# B&R Automation Studio project EFI (part 3)

### Hardware
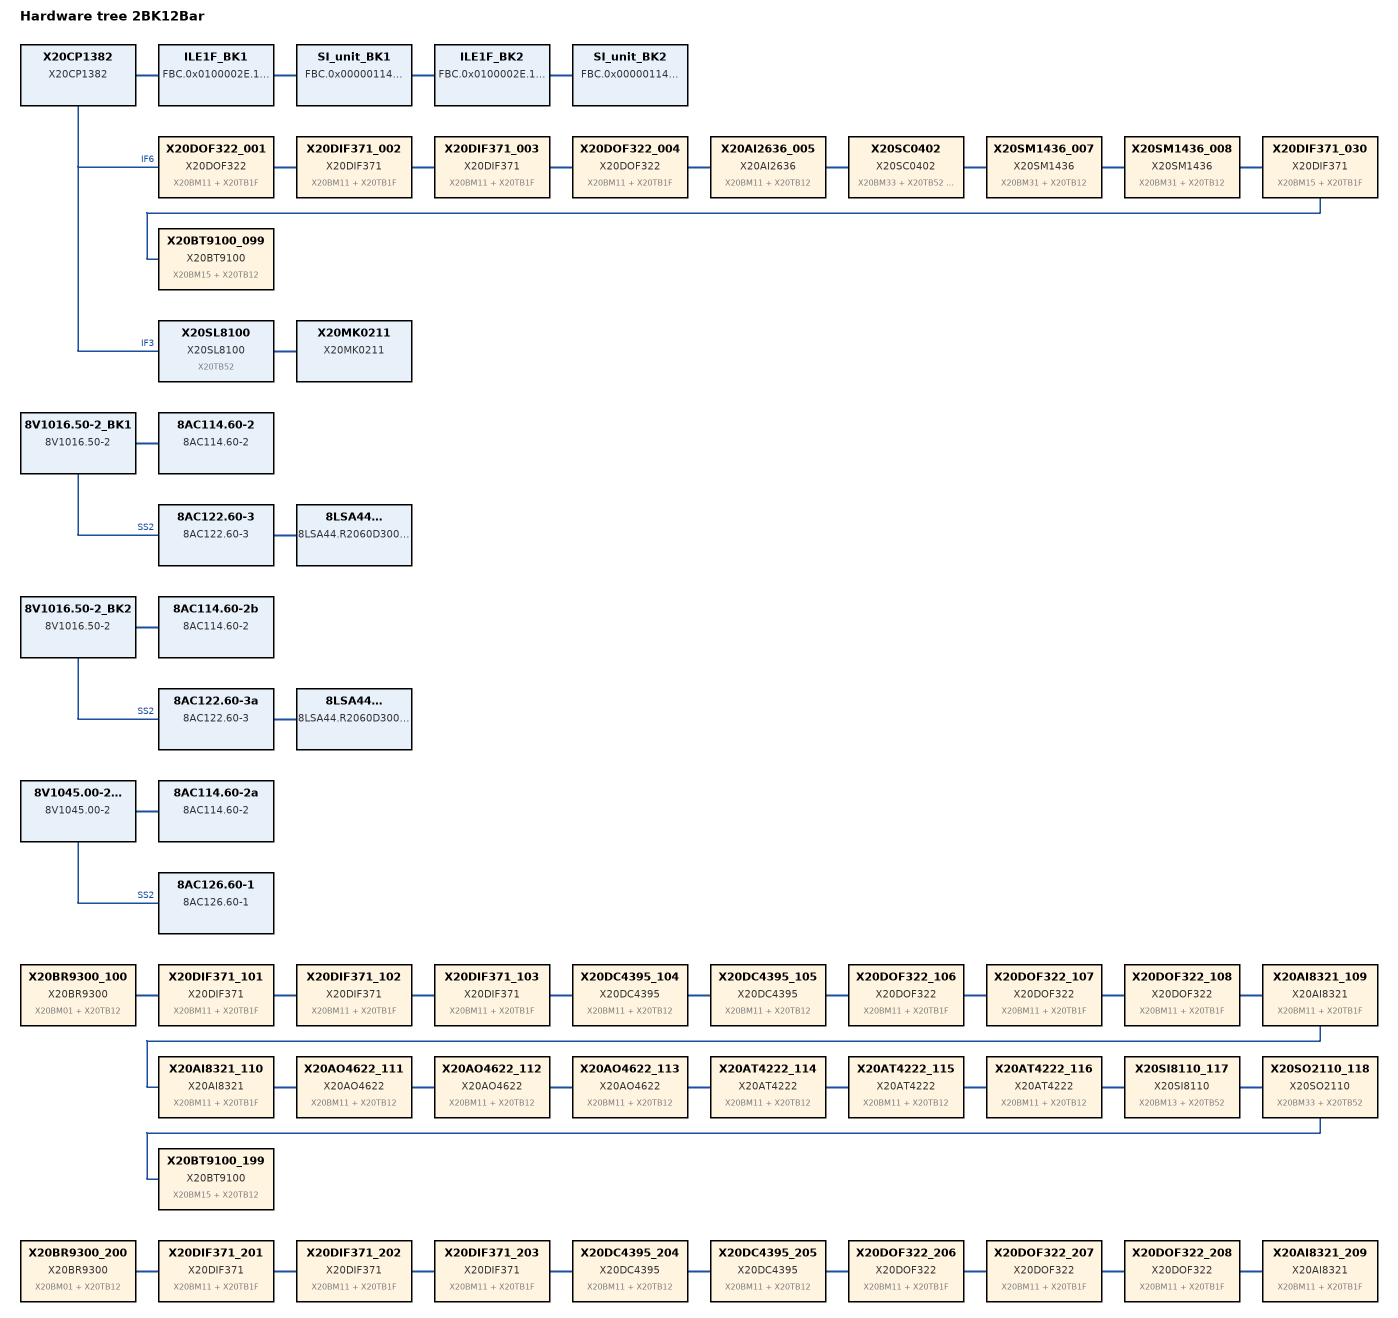
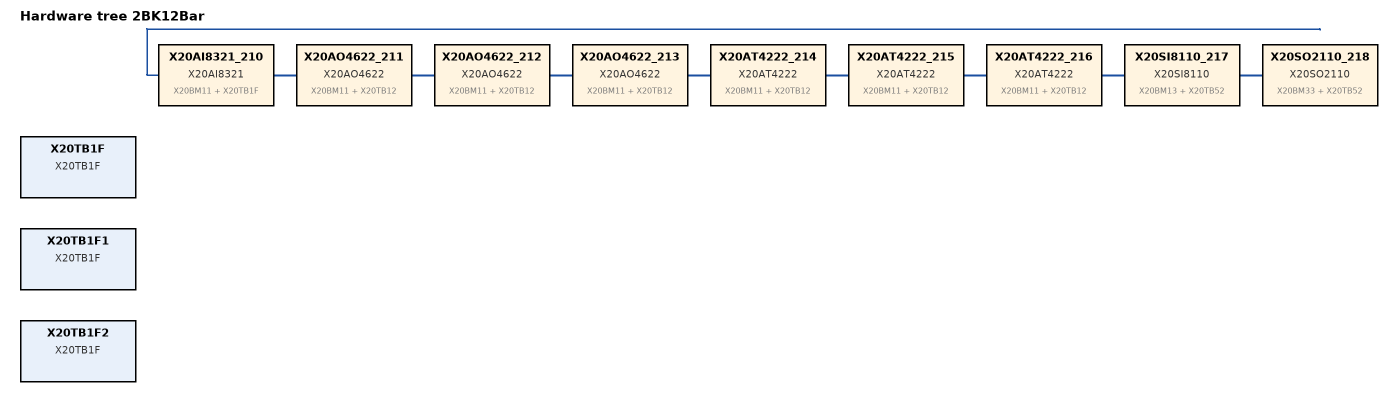
```
8AC114.60-2 : 8AC114.60-2 v1.0.0.8  [SS -> 8V1016.50-2_BK1.SS1; PLK1 -> 8AC114.60-2a.PLK2 (NodeNumber=2) [Cable Type=PowerlinkCable, Length=10, Version=1.0.0.3]; PLK2 -> 8AC114.60-2b.PLK1 (NodeNumber=2) [Cable Type=PowerlinkCable, Length=10, Version=1.0.0.3]]
8AC114.60-2a : 8AC114.60-2 v1.0.0.8  [SS -> 8V1045.00-2_BELT.SS1; PLK1 -> X20SL8100.PLK2 (NodeNumber=1) [Cable Type=PowerlinkCable, Length=10, Version=1.0.0.3]; PLK2 -> 8AC114.60-2.PLK1 (NodeNumber=1) [Cable Type=PowerlinkCable, Length=10, Version=1.0.0.3]]
8AC114.60-2b : 8AC114.60-2 v1.0.0.8  [SS -> 8V1016.50-2_BK2.SS1; PLK1 -> 8AC114.60-2.PLK2 (NodeNumber=3) [Cable Type=PowerlinkCable, Length=10, Version=1.0.0.3]]
8AC122.60-3 : 8AC122.60-3 v2.2.0.0  [SS -> 8V1016.50-2_BK1.SS2]
8AC122.60-3a : 8AC122.60-3 v2.2.0.0  [SS -> 8V1016.50-2_BK2.SS2]
8AC126.60-1 : 8AC126.60-1 v2.2.0.0  [SS -> 8V1045.00-2_BELT.SS2]
8LSA44.R2060D300-3 : 8LSA44.R2060D300-3 v2.2.0.0  [EC -> 8AC122.60-3.EC; MT -> 8V1016.50-2_BK1.MT1]
8LSA44.R2060D300-3a : 8LSA44.R2060D300-3 v2.2.0.0  [EC -> 8AC122.60-3a.EC; MT -> 8V1016.50-2_BK2.MT1]
8V1016.50-2_BK1 : 8V1016.50-2 v2.2.0.0
  SinglePhaseOperation = on
  BothEndSwitchesAreNormallyOpen_r1 = on
  QuickStopIsNormallyOpen_r1 = on
8V1016.50-2_BK2 : 8V1016.50-2 v2.2.0.0
  SinglePhaseOperation = on
  BothEndSwitchesAreNormallyOpen_r1 = on
  QuickStopIsNormallyOpen_r1 = on
8V1045.00-2_BELT : 8V1045.00-2 v2.2.0.0
ILE1F_BK1 : FBC.0x0100002E.1.SEILE1F_0110E v1.10 (OrderNumber=ILE1F)  [CAN1 -> X20CP1382.IF7 (NodeNumber=5)]
  p1403_transmissionselection = 1
  plifeguarding_guardtime = 500
  plifeguarding_retryfactor = 10
  p3001_parametername = mandatory
  p3001_objecttype = 9
  p3001_subnumber = 0x3
  p3001_parametervalue = 
  p3001_objflags = 0
  p3001sub0_parametername = number of entries
  p3001sub0_objecttype = 7
  p3001sub0_datatype = 5
  p3001sub0_accesstype = ro
  p3001sub0_pdomapping = 0
  p3001sub1_parametername = Config.PrgNo
  p3001sub1_objecttype = 7
  p3001sub1_datatype = 7
  p3001sub1_lowlimit = 
  p3001sub1_highlimit = 
  p3001sub1_accesstype = ro
  p3001sub1_pdomapping = 0
  p3001sub2_parametername = Config.PrgVer
  p3001sub2_objecttype = 7
  p3001sub2_datatype = 7
  p3001sub2_lowlimit = 
  p3001sub2_highlimit = 
  p3001sub2_accesstype = ro
  p3001sub2_pdomapping = 0
  p300b_parametername = system settings
  p300b_objecttype = 9
  p300b_subnumber = 0x7
  p300b_parametervalue = 
  p300b_objflags = 0
  p300bsub0_parametername = number of entries
  p300bsub0_objecttype = 7
  p300bsub0_datatype = 5
  p300bsub0_accesstype = ro
  p300bsub0_pdomapping = 0
  p300bsub1_parametername = Settings.name1
  p300bsub1_objecttype = 7
  p300bsub1_datatype = 7
  p300bsub1_lowlimit = 
  p300bsub1_highlimit = 
  p300bsub1_accesstype = rw
  p300bsub1_pdomapping = 0
  p300bsub1_parametervalue = 
  p300bsub1_objflags = 0
  p300bsub2_parametername = Settings.name2
  p300bsub2_objecttype = 7
  p300bsub2_datatype = 7
  p300bsub2_lowlimit = 
  p300bsub2_highlimit = 
  p300bsub2_accesstype = rw
  p300bsub2_pdomapping = 0
  p300bsub2_parametervalue = 
  p300bsub2_objflags = 0
  p300bsub6_parametername = Commands.eeprSave
  p300bsub6_objecttype = 7
  p300bsub6_datatype = 6
  p300bsub6_lowlimit = 
  p300bsub6_highlimit = 
  p300bsub6_accesstype = rw
  p300bsub6_pdomapping = 0
  p300bsub6_parametervalue = 1
  p300bsub6_objflags = 0
  p300bsub7_parametername = Commands.stateSave
  p300bsub7_objecttype = 7
  p300bsub7_datatype = 6
  p300bsub7_lowlimit = 
  p300bsub7_highlimit = 
  p300bsub7_accesstype = ro
  p300bsub7_pdomapping = 0
  p300bsub8_parametername = Commands.default
  p300bsub8_objecttype = 7
  p300bsub8_datatype = 6
  p300bsub8_lowlimit = 
  p300bsub8_highlimit = 
  p300bsub8_accesstype = rw
  p300bsub8_pdomapping = 0
  p300bsub8_parametervalue = 
  p300bsub8_objflags = 0
  p300bsub9_parametername = Commands.stateDef
  p300bsub9_objecttype = 7
  p300bsub9_datatype = 6
  p300bsub9_lowlimit = 
  p300bsub9_highlimit = 
  p300bsub9_accesstype = ro
  p300bsub9_pdomapping = 0
  p300f_parametername = controller  settings
  p300f_objecttype = 9
  p300f_subnumber = 0xE
  p300f_parametervalue = 
  p300f_objflags = 0
  p300fsub0_parametername = number of entries
  p300fsub0_objecttype = 7
  p300fsub0_datatype = 5
  p300fsub0_accesstype = ro
  p300fsub0_pdomapping = 0
  p300fsub1_parametername = Config.I_nomDrv
  p300fsub1_objecttype = 7
  p300fsub1_datatype = 6
  p300fsub1_accesstype = ro
  p300fsub1_pdomapping = 0
  p300fsub2_parametername = Config.I_maxDrv
  p300fsub2_objecttype = 7
  p300fsub2_datatype = 6
  p300fsub2_accesstype = ro
  p300fsub2_pdomapping = 0
  p300fsub3_parametername = Settings.I_max
  p300fsub3_objecttype = 7
  p300fsub3_datatype = 6
  p300fsub3_accesstype = rw
  p300fsub3_pdomapping = 0
  p300fsub3_parametervalue = 60
  p300fsub3_objflags = 0
  p300fsub5_parametername = Settings.I_maxBlk
  p300fsub5_objecttype = 7
  p300fsub5_datatype = 6
  p300fsub5_lowlimit = 
  p300fsub5_highlimit = 
  p300fsub5_accesstype = rw
  p300fsub5_pdomapping = 0
  p300fsub5_parametervalue = 20
  p300fsub5_objflags = 0
  p300fsub7_parametername = Settings.p_maxDiff
  p300fsub7_objecttype = 7
  p300fsub7_datatype = 6
  p300fsub7_lowlimit = 
  p300fsub7_highlimit = 
  p300fsub7_accesstype = rw
  p300fsub7_pdomapping = 0
  p300fsub7_parametervalue = 24
  p300fsub7_objflags = 0
  p300fsub8_parametername = Control.KPn
  p300fsub8_objecttype = 7
  p300fsub8_datatype = 6
  p300fsub8_lowlimit = 
  p300fsub8_highlimit = 
  p300fsub8_accesstype = rw
  p300fsub8_pdomapping = 0
  p300fsub8_parametervalue = 60
  p300fsub8_objflags = 0
  p300fsub9_parametername = Control.TNn
  p300fsub9_objecttype = 7
  p300fsub9_datatype = 6
  p300fsub9_lowlimit = 
  p300fsub9_highlimit = 
  p300fsub9_accesstype = rw
  p300fsub9_pdomapping = 0
  p300fsub9_parametervalue = 10000
  p300fsub9_objflags = 0
  p300fsuba_parametername = Control.KPp
  p300fsuba_objecttype = 7
  p300fsuba_datatype = 6
  p300fsuba_lowlimit = 
  p300fsuba_highlimit = 
  p300fsuba_accesstype = rw
  p300fsuba_pdomapping = 0
  p300fsuba_parametervalue = 300
  p300fsuba_objflags = 0
  p300fsubb_parametername = Control.KFPp
  p300fsubb_objecttype = 7
  p300fsubb_datatype = 6
  p300fsubb_lowlimit = 
  p300fsubb_highlimit = 
  p300fsubb_accesstype = rw
  p300fsubb_pdomapping = 0
  p300fsubb_parametervalue = 32767
  p300fsubb_objflags = 0
  p300fsubc_parametername = Settings.T_block
  p300fsubc_objecttype = 7
  p300fsubc_datatype = 6
  p300fsubc_lowlimit = 
  p300fsubc_highlimit = 
  p300fsubc_accesstype = rw
  p300fsubc_pdomapping = 0
  p300fsubc_parametervalue = 100
  p300fsubc_objflags = 0
  p300fsubd_parametername = Status.p_difPeak
  p300fsubd_objecttype = 7
  p300fsubd_datatype = 7
  p300fsubd_lowlimit = 
  p300fsubd_highlimit = 
  p300fsubd_accesstype = rw
  p300fsubd_pdomapping = 0
  p300fsubd_parametervalue = 
  p300fsubd_objflags = 0
  p300fsubf_parametername = Settings.p_win
  p300fsubf_objecttype = 7
  p300fsubf_datatype = 6
  p300fsubf_lowlimit = 
  p300fsubf_highlimit = 
  p300fsubf_accesstype = rw
  p300fsubf_pdomapping = 0
  p300fsubf_parametervalue = 1
  p300fsubf_objflags = 0
  p300fsub10_parametername = Settings.p_winTime
  p300fsub10_objecttype = 7
  p300fsub10_datatype = 6
  p300fsub10_lowlimit = 
  p300fsub10_highlimit = 
  p300fsub10_accesstype = rw
  p300fsub10_pdomapping = 0
  p300fsub10_parametervalue = 0
  p300fsub10_objflags = 0
  p3016_parametername = rs485
  p3016_objecttype = 9
  p3016_subnumber = 0x4
  p3016_parametervalue = 
  p3016_objflags = 0
  p3016sub0_parametername = number of entries
  p3016sub0_objecttype = 7
  p3016sub0_datatype = 5
  p3016sub0_accesstype = ro
  p3016sub0_pdomapping = 0
  p3016sub1_parametername = RS485.serBaud
  p3016sub1_objecttype = 7
  p3016sub1_datatype = 6
  p3016sub1_lowlimit = 
  p3016sub1_highlimit = 
  p3016sub1_accesstype = rw
  p3016sub1_pdomapping = 0
  p3016sub1_parametervalue = 
  p3016sub1_objflags = 0
  p3016sub2_parametername = RS485.serAdr
  p3016sub2_objecttype = 7
  p3016sub2_datatype = 6
  p3016sub2_lowlimit = 
  p3016sub2_highlimit = 
  p3016sub2_accesstype = rw
  p3016sub2_pdomapping = 0
  p3016sub2_parametervalue = 
  p3016sub2_objflags = 0
  p3016sub3_parametername = RS485.serFormat
  p3016sub3_objecttype = 7
  p3016sub3_datatype = 6
  p3016sub3_lowlimit = 
  p3016sub3_highlimit = 
  p3016sub3_accesstype = rw
  p3016sub3_pdomapping = 0
  p3016sub3_parametervalue = 
  p3016sub3_objflags = 0
  p3017_parametername = can
  p3017_objecttype = 9
  p3017_subnumber = 0x3
  p3017_parametervalue = 
  p3017_objflags = 0
  p3017sub0_parametername = number of entries
  p3017sub0_objecttype = 7
  p3017sub0_datatype = 5
  p3017sub0_accesstype = ro
  p3017sub0_pdomapping = 0
  p3017sub2_parametername = CAN.canAddr
  p3017sub2_objecttype = 7
  p3017sub2_datatype = 6
  p3017sub2_lowlimit = 
  p3017sub2_highlimit = 
  p3017sub2_accesstype = rw
  p3017sub2_pdomapping = 0
  p3017sub2_parametervalue = 
  p3017sub2_objflags = 0
  p3017sub3_parametername = CAN.canBaud
  p3017sub3_objecttype = 7
  p3017sub3_datatype = 6
  p3017sub3_lowlimit = 
  p3017sub3_highlimit = 
  p3017sub3_accesstype = rw
  p3017sub3_pdomapping = 0
  p3017sub3_parametervalue = 
  p3017sub3_objflags = 0
  p301c_parametername = settings1
  p301c_objecttype = 9
  p301c_subnumber = 0xF
  p301c_parametervalue = 
  p301c_objflags = 0
  p301csub0_parametername = number of entries
  p301csub0_objecttype = 7
  p301csub0_datatype = 5
  p301csub0_accesstype = ro
  p301csub0_pdomapping = 0
  p301csub3_parametername = Status.xMode_act
  p301csub3_objecttype = 7
  p301csub3_datatype = 6
  p301csub3_lowlimit = 
  p301csub3_highlimit = 
  p301csub3_accesstype = ro
  p301csub3_pdomapping = 0
  p301csub6_parametername = Motion.invertDir
  p301csub6_objecttype = 7
  p301csub6_datatype = 6
  p301csub6_lowlimit = 
  p301csub6_highlimit = 
  p301csub6_accesstype = rw
  p301csub6_pdomapping = 0
  p301csub6_parametervalue = 0
  p301csub6_objflags = 0
  p301csuba_parametername = Status.WarnSig
  p301csuba_objecttype = 7
  p301csuba_datatype = 6
  p301csuba_lowlimit = 
  p301csuba_highlimit = 
  p301csuba_accesstype = ro
  p301csuba_pdomapping = 0
  p301csubb_parametername = Settings.WarnOvrun
  p301csubb_objecttype = 7
  p301csubb_datatype = 6
  p301csubb_lowlimit = 
  p301csubb_highlimit = 
  p301csubb_accesstype = rw
  p301csubb_pdomapping = 0
  p301csubb_parametervalue = 0
  p301csubb_objflags = 0
  p301csubd_parametername = Settings.SignEnabl
  p301csubd_objecttype = 7
  p301csubd_datatype = 6
  p301csubd_lowlimit = 
  p301csubd_highlimit = 
  p301csubd_accesstype = rw
  p301csubd_pdomapping = 0
  p301csubd_parametervalue = 3
  p301csubd_objflags = 0
  p301csube_parametername = Settings.SignLevel
  p301csube_objecttype = 7
  p301csube_datatype = 6
  p301csube_lowlimit = 
  p301csube_highlimit = 
  p301csube_accesstype = rw
  p301csube_pdomapping = 0
  p301csube_parametervalue = 0
  p301csube_objflags = 0
  p301csubf_parametername = Status.Sign_SR
  p301csubf_objecttype = 7
  p301csubf_datatype = 6
  p301csubf_lowlimit = 
  p301csubf_highlimit = 
  p301csubf_accesstype = ro
  p301csubf_pdomapping = 0
  p301csub11_parametername = Status.FltSig
  p301csub11_objecttype = 7
  p301csub11_datatype = 7
  p301csub11_lowlimit = 
  p301csub11_highlimit = 
  p301csub11_accesstype = ro
  p301csub11_pdomapping = 0
  p301csub12_parametername = Status.FltSig_SR
  p301csub12_objecttype = 7
  p301csub12_datatype = 7
  p301csub12_lowlimit = 
  p301csub12_highlimit = 
  p301csub12_accesstype = ro
  p301csub12_pdomapping = 0
  p301csub13_parametername = Status.action_st
  p301csub13_objecttype = 7
  p301csub13_datatype = 6
  p301csub13_lowlimit = 
  p301csub13_highlimit = 
  p301csub13_accesstype = ro
  p301csub13_pdomapping = 0
  p301csub15_parametername = Motion.dec_Stop
  p301csub15_objecttype = 7
  p301csub15_datatype = 7
  p301csub15_lowlimit = 
  p301csub15_highlimit = 
  p301csub15_accesstype = rw
  p301csub15_pdomapping = 0
  p301csub15_parametervalue = 4960
  p301csub15_objflags = 0
  p301csub18_parametername = Settings.Flt_pDiff
  p301csub18_objecttype = 7
  p301csub18_datatype = 6
  p301csub18_lowlimit = 
  p301csub18_highlimit = 
  p301csub18_accesstype = rw
  p301csub18_pdomapping = 0
  p301csub18_parametervalue = 3
  p301csub18_objflags = 0
  p301d_parametername = settings2
  p301d_objecttype = 9
  p301d_subnumber = 0x4
  p301d_parametervalue = 
  p301d_objflags = 0
  p301dsub0_parametername = number of entries
  p301dsub0_objecttype = 7
  p301dsub0_datatype = 5
  p301dsub0_accesstype = ro
  p301dsub0_pdomapping = 0
  p301dsub2_parametername = Config.ResolutM
  p301dsub2_objecttype = 7
  p301dsub2_datatype = 6
  p301dsub2_accesstype = ro
  p301dsub2_pdomapping = 0
  p301dsub17_parametername = Motion.v_target0
  p301dsub17_objecttype = 7
  p301dsub17_datatype = 6
  p301dsub17_accesstype = rw
  p301dsub17_pdomapping = 0
  p301dsub17_parametervalue = 1000
  p301dsub17_objflags = 0
  p301dsub1a_parametername = Motion.acc
  p301dsub1a_objecttype = 7
  p301dsub1a_datatype = 7
  p301dsub1a_lowlimit = 
  p301dsub1a_highlimit = 
  p301dsub1a_accesstype = rw
  p301dsub1a_pdomapping = 0
  p301dsub1a_parametervalue = 2442
  p301dsub1a_objflags = 0
  p301e_parametername = pdo data
  p301e_objecttype = 9
  p301e_subnumber = 0xC
  p301e_parametervalue = 
  p301e_objflags = 0
  p301esub0_parametername = number of entries
  p301esub0_objecttype = 7
  p301esub0_datatype = 5
  p301esub0_accesstype = ro
  p301esub0_pdomapping = 0
  p301esubb_parametername = Status.ModeError
  p301esubb_objecttype = 7
  p301esubb_datatype = 6
  p301esubb_lowlimit = 
  p301esubb_highlimit = 
  p301esubb_accesstype = ro
  p301esubb_pdomapping = 0
  p301f_parametername = status
  p301f_objecttype = 9
  p301f_subnumber = 0x11
  p301f_parametervalue = 
  p301f_objflags = 0
  p301fsub0_parametername = number of entries
  p301fsub0_objecttype = 7
  p301fsub0_datatype = 5
  p301fsub0_accesstype = ro
  p301fsub0_pdomapping = 0
  p301fsub1_parametername = Status.v_ref
  p301fsub1_objecttype = 7
  p301fsub1_datatype = 4
  p301fsub1_lowlimit = 
  p301fsub1_highlimit = 
  p301fsub1_accesstype = ro
  p301fsub1_pdomapping = 0
  p301fsub2_parametername = Status.v_act
  p301fsub2_objecttype = 7
  p301fsub2_datatype = 4
  p301fsub2_lowlimit = 
  p301fsub2_highlimit = 
  p301fsub2_accesstype = ro
  p301fsub2_pdomapping = 0
  p301fsub5_parametername = Status.p_ref
  p301fsub5_objecttype = 7
  p301fsub5_datatype = 4
  p301fsub5_lowlimit = 
  p301fsub5_highlimit = 
  p301fsub5_accesstype = ro
  p301fsub5_pdomapping = 0
  p301fsub6_parametername = Status.p_act
  p301fsub6_objecttype = 7
  p301fsub6_datatype = 4
  p301fsub6_lowlimit = 
  p301fsub6_highlimit = 
  p301fsub6_accesstype = ro
  p301fsub6_pdomapping = 0
  p301fsub7_parametername = Status.p_dif
  p301fsub7_objecttype = 7
  p301fsub7_datatype = 4
  p301fsub7_lowlimit = 
  p301fsub7_highlimit = 
  p301fsub7_accesstype = ro
  p301fsub7_pdomapping = 0
  p301fsub8_parametername = Status.n_ref
  p301fsub8_objecttype = 7
  p301fsub8_datatype = 3
  p301fsub8_lowlimit = 
  p301fsub8_highlimit = 
  p301fsub8_accesstype = ro
  p301fsub8_pdomapping = 0
  p301fsub9_parametername = Status.n_act
  p301fsub9_objecttype = 7
  p301fsub9_datatype = 3
  p301fsub9_lowlimit = 
  p301fsub9_highlimit = 
  p301fsub9_accesstype = ro
  p301fsub9_pdomapping = 0
  p301fsubc_parametername = Status.I_act
  p301fsubc_objecttype = 7
  p301fsubc_datatype = 3
  p301fsubc_lowlimit = 
  p301fsubc_highlimit = 
  p301fsubc_accesstype = ro
  p301fsubc_pdomapping = 0
  p301fsub14_parametername = Status.UDC_act
  p301fsub14_objecttype = 7
  p301fsub14_datatype = 6
  p301fsub14_lowlimit = 
  p301fsub14_highlimit = 
  p301fsub14_accesstype = ro
  p301fsub14_pdomapping = 0
  p301fsub19_parametername = Status.TPA_act
  p301fsub19_objecttype = 7
  p301fsub19_datatype = 6
  p301fsub19_lowlimit = 
  p301fsub19_highlimit = 
  p301fsub19_accesstype = ro
  p301fsub19_pdomapping = 0
  p301fsub1c_parametername = Status.v_pref
  p301fsub1c_objecttype = 7
  p301fsub1c_datatype = 4
  p301fsub1c_lowlimit = 
  p301fsub1c_highlimit = 
  p301fsub1c_accesstype = ro
  p301fsub1c_pdomapping = 0
  p301fsub1e_parametername = Status.p_target
  p301fsub1e_objecttype = 7
  p301fsub1e_datatype = 4
  p301fsub1e_lowlimit = 
  p301fsub1e_highlimit = 
  p301fsub1e_accesstype = ro
  p301fsub1e_pdomapping = 0
  p301fsub1f_parametername = Status.p_profile
  p301fsub1f_objecttype = 7
  p301fsub1f_datatype = 4
  p301fsub1f_lowlimit = 
  p301fsub1f_highlimit = 
  p301fsub1f_accesstype = ro
  p301fsub1f_pdomapping = 0
  p301fsub23_parametername = Status.n_profile
  p301fsub23_objecttype = 7
  p301fsub23_datatype = 3
  p301fsub23_lowlimit = 
  p301fsub23_highlimit = 
  p301fsub23_accesstype = ro
  p301fsub23_pdomapping = 0
  p301fsub26_parametername = Status.n_target
  p301fsub26_objecttype = 7
  p301fsub26_datatype = 3
  p301fsub26_lowlimit = 
  p301fsub26_highlimit = 
  p301fsub26_accesstype = ro
  p301fsub26_pdomapping = 0
  p301fsub2d_parametername = Status.n_pref
  p301fsub2d_objecttype = 7
  p301fsub2d_datatype = 3
  p301fsub2d_lowlimit = 
  p301fsub2d_highlimit = 
  p301fsub2d_accesstype = ro
  p301fsub2d_pdomapping = 0
  p3020_parametername = error
  p3020_objecttype = 9
  p3020_subnumber = 0x5
  p3020_parametervalue = 
  p3020_objflags = 0
  p3020sub0_parametername = number of entries
  p3020sub0_objecttype = 7
  p3020sub0_datatype = 5
  p3020sub0_accesstype = ro
  p3020sub0_pdomapping = 0
  p3020sub1_parametername = ErrorMemAvailable
  p3020sub1_objecttype = 7
  p3020sub1_datatype = 6
  p3020sub1_lowlimit = 
  p3020sub1_highlimit = 
  p3020sub1_accesstype = ro
  p3020sub1_pdomapping = 0
  p3020sub2_parametername = Commands.del_err
  p3020sub2_objecttype = 7
  p3020sub2_datatype = 6
  p3020sub2_lowlimit = 
  p3020sub2_highlimit = 
  p3020sub2_accesstype = rw
  p3020sub2_pdomapping = 0
  p3020sub2_parametervalue = 
  p3020sub2_objflags = 0
  p3020sub6_parametername = PowerOnCount
  p3020sub6_objecttype = 7
  p3020sub6_datatype = 7
  p3020sub6_lowlimit = 
  p3020sub6_highlimit = 
  p3020sub6_accesstype = ro
  p3020sub6_pdomapping = 0
  p3020sub7_parametername = Status.StopFault
  p3020sub7_objecttype = 7
  p3020sub7_datatype = 6
  p3020sub7_lowlimit = 
  p3020sub7_highlimit = 
  p3020sub7_accesstype = ro
  p3020sub7_pdomapping = 0
  p3021_parametername = io
  p3021_objecttype = 9
  p3021_subnumber = 0x4
  p3021_parametervalue = 
  p3021_objflags = 0
  p3021sub0_parametername = number of entries
  p3021sub0_objecttype = 7
  p3021sub0_datatype = 5
  p3021sub0_accesstype = ro
  p3021sub0_pdomapping = 0
  p3021sub1_parametername = I/O.IO_act
  p3021sub1_objecttype = 7
  p3021sub1_datatype = 6
  p3021sub1_lowlimit = 
  p3021sub1_highlimit = 
  p3021sub1_accesstype = rw
  p3021sub1_pdomapping = 0
  p3021sub1_parametervalue = 
  p3021sub1_objflags = 0
  p3021sub7_parametername = Commands.brake
  p3021sub7_objecttype = 7
  p3021sub7_datatype = 6
  p3021sub7_lowlimit = 
  p3021sub7_highlimit = 
  p3021sub7_accesstype = rw
  p3021sub7_pdomapping = 0
  p3021sub7_parametervalue = 
  p3021sub7_objflags = 0
  p3021sub8_parametername = Status.brake
  p3021sub8_objecttype = 7
  p3021sub8_datatype = 6
  p3021sub8_lowlimit = 
  p3021sub8_highlimit = 
  p3021sub8_accesstype = ro
  p3021sub8_pdomapping = 0
  p3022_parametername = io definitions
  p3022_objecttype = 9
  p3022_subnumber = 0x6
  p3022_parametervalue = 
  p3022_objflags = 0
  p3022sub0_parametername = number of entries
  p3022sub0_objecttype = 7
  p3022sub0_datatype = 5
  p3022sub0_accesstype = ro
  p3022sub0_pdomapping = 0
  p3022sub1_parametername = I/O.IO0_def
  p3022sub1_objecttype = 7
  p3022sub1_datatype = 6
  p3022sub1_lowlimit = 
  p3022sub1_highlimit = 
  p3022sub1_accesstype = rw
  p3022sub1_pdomapping = 0
  p3022sub1_parametervalue = 0
  p3022sub1_objflags = 0
  p3022sub2_parametername = I/O.IO1_def
  p3022sub2_objecttype = 7
  p3022sub2_datatype = 6
  p3022sub2_lowlimit = 
  p3022sub2_highlimit = 
  p3022sub2_accesstype = rw
  p3022sub2_pdomapping = 0
  p3022sub2_parametervalue = 0
  p3022sub2_objflags = 0
  p3022sub3_parametername = I/O.IO2_def
  p3022sub3_objecttype = 7
  p3022sub3_datatype = 6
  p3022sub3_lowlimit = 
  p3022sub3_highlimit = 
  p3022sub3_accesstype = rw
  p3022sub3_pdomapping = 0
  p3022sub3_parametervalue = 0
  p3022sub3_objflags = 0
  p3022sub4_parametername = I/O.IO3_def
  p3022sub4_objecttype = 7
  p3022sub4_datatype = 6
  p3022sub4_lowlimit = 
  p3022sub4_highlimit = 
  p3022sub4_accesstype = rw
  p3022sub4_pdomapping = 0
  p3022sub4_parametervalue = 
  p3022sub4_objflags = 0
  p3022sub7_parametername = I/O.progDelay
  p3022sub7_objecttype = 7
  p3022sub7_datatype = 6
  p3022sub7_lowlimit = 
  p3022sub7_highlimit = 
  p3022sub7_accesstype = rw
  p3022sub7_pdomapping = 0
  p3022sub7_parametervalue = 
  p3022sub7_objflags = 0
  p3023_parametername = ptp
  p3023_objecttype = 9
  p3023_subnumber = 0x6
  p3023_parametervalue = 
  p3023_objflags = 0
  p3023sub0_parametername = number of entries
  p3023sub0_objecttype = 7
  p3023sub0_datatype = 5
  p3023sub0_accesstype = ro
  p3023sub0_pdomapping = 0
  p3023sub1_parametername = PTP.p_absPTP
  p3023sub1_objecttype = 7
  p3023sub1_datatype = 4
  p3023sub1_lowlimit = 
  p3023sub1_highlimit = 
  p3023sub1_accesstype = rw
  p3023sub1_pdomapping = 0
  p3023sub1_parametervalue = 
  p3023sub1_objflags = 0
  p3023sub2_parametername = PTP.StatePTP
  p3023sub2_objecttype = 7
  p3023sub2_datatype = 6
  p3023sub2_lowlimit = 
  p3023sub2_highlimit = 
  p3023sub2_accesstype = ro
  p3023sub2_pdomapping = 0
  p3023sub3_parametername = PTP.p_relPTP
  p3023sub3_objecttype = 7
  p3023sub3_datatype = 4
  p3023sub3_lowlimit = 
  p3023sub3_highlimit = 
  p3023sub3_accesstype = rw
  p3023sub3_pdomapping = 0
  p3023sub3_parametervalue = 
  p3023sub3_objflags = 0
  p3023sub4_parametername = PTP.continue
  p3023sub4_objecttype = 7
  p3023sub4_datatype = 6
  p3023sub4_lowlimit = 
  p3023sub4_highlimit = 
  p3023sub4_accesstype = rw
  p3023sub4_pdomapping = 0
  p3023sub4_parametervalue = 
  p3023sub4_objflags = 0
  p3023sub5_parametername = PTP.v_tarPTP
  p3023sub5_objecttype = 7
  p3023sub5_datatype = 6
  p3023sub5_accesstype = rw
  p3023sub5_pdomapping = 0
  p3023sub5_parametervalue = 
  p3023sub5_objflags = 0
  p3024_parametername = vel
  p3024_objecttype = 9
  p3024_subnumber = 0x3
  p3024_parametervalue = 
  p3024_objflags = 0
  p3024sub0_parametername = number of entries
  p3024sub0_objecttype = 7
  p3024sub0_datatype = 5
  p3024sub0_accesstype = ro
  p3024sub0_pdomapping = 0
  p3024sub1_parametername = VEL.velocity
  p3024sub1_objecttype = 7
  p3024sub1_datatype = 3
  p3024sub1_accesstype = rw
  p3024sub1_pdomapping = 0
  p3024sub1_parametervalue = 
  p3024sub1_objflags = 0
  p3024sub2_parametername = VEL.stateVEL
  p3024sub2_objecttype = 7
  p3024sub2_datatype = 6
  p3024sub2_lowlimit = 
  p3024sub2_highlimit = 
  p3024sub2_accesstype = ro
  p3024sub2_pdomapping = 0
  p3028_parametername = homing
  p3028_objecttype = 9
  p3028_subnumber = 0xB
  p3028_parametervalue = 
  p3028_objflags = 0
  p3028sub0_parametername = number of entries
  p3028sub0_objecttype = 7
  p3028sub0_datatype = 5
  p3028sub0_accesstype = ro
  p3028sub0_pdomapping = 0
  p3028sub1_parametername = Homing.startHome
  p3028sub1_objecttype = 7
  p3028sub1_datatype = 6
  p3028sub1_lowlimit = 
  p3028sub1_highlimit = 
  p3028sub1_accesstype = rw
  p3028sub1_pdomapping = 0
  p3028sub1_parametervalue = 
  p3028sub1_objflags = 0
  p3028sub2_parametername = Homing.stateHome
  p3028sub2_objecttype = 7
  p3028sub2_datatype = 6
  p3028sub2_lowlimit = 
  p3028sub2_highlimit = 
  p3028sub2_accesstype = ro
  p3028sub2_pdomapping = 0
  p3028sub3_parametername = Homing.startSetp
  p3028sub3_objecttype = 7
  p3028sub3_datatype = 4
  p3028sub3_lowlimit = 
  p3028sub3_highlimit = 
  p3028sub3_accesstype = rw
  p3028sub3_pdomapping = 0
  p3028sub3_parametervalue = 
  p3028sub3_objflags = 0
  p3028sub4_parametername = Homing.v_Home
  p3028sub4_objecttype = 7
  p3028sub4_datatype = 6
  p3028sub4_accesstype = rw
  p3028sub4_pdomapping = 0
  p3028sub4_parametervalue = 
  p3028sub4_objflags = 0
  p3028sub5_parametername = Homing.v_outHome
  p3028sub5_objecttype = 7
  p3028sub5_datatype = 6
  p3028sub5_accesstype = rw
  p3028sub5_pdomapping = 0
  p3028sub5_parametervalue = 
  p3028sub5_objflags = 0
  p3028sub6_parametername = Homing.p_outHome
  p3028sub6_objecttype = 7
  p3028sub6_datatype = 4
  p3028sub6_lowlimit = 
  p3028sub6_highlimit = 
  p3028sub6_accesstype = rw
  p3028sub6_pdomapping = 0
  p3028sub6_parametervalue = 
  p3028sub6_objflags = 0
  p3028sub7_parametername = Homing.p_disHome
  p3028sub7_objecttype = 7
  p3028sub7_datatype = 4
  p3028sub7_lowlimit = 
  p3028sub7_highlimit = 
  p3028sub7_accesstype = rw
  p3028sub7_pdomapping = 0
  p3028sub7_parametervalue = 
  p3028sub7_objflags = 0
  p3028sub9_parametername = Homing.RefSwMod
  p3028sub9_objecttype = 7
  p3028sub9_datatype = 6
  p3028sub9_lowlimit = 
  p3028sub9_highlimit = 
  p3028sub9_accesstype = rw
  p3028sub9_pdomapping = 0
  p3028sub9_parametervalue = 
  p3028sub9_objflags = 0
  p3028subb_parametername = Homing.RefAppPos
  p3028subb_objecttype = 7
  p3028subb_datatype = 4
  p3028subb_lowlimit = 
  p3028subb_highlimit = 
  p3028subb_accesstype = rw
  p3028subb_pdomapping = 0
  p3028subb_parametervalue = 
  p3028subb_objflags = 0
  p3028subd_parametername = Homing.refError
  p3028subd_objecttype = 7
  p3028subd_datatype = 6
  p3028subd_lowlimit = 
  p3028subd_highlimit = 
  p3028subd_accesstype = ro
  p3028subd_pdomapping = 0
  p3029_parametername = manual
  p3029_objecttype = 9
  p3029_subnumber = 0x7
  p3029_parametervalue = 
  p3029_objflags = 0
  p3029sub0_parametername = number of entries
  p3029sub0_objecttype = 7
  p3029sub0_datatype = 5
  p3029sub0_accesstype = ro
  p3029sub0_pdomapping = 0
  p3029sub1_parametername = Manual.startMan
  p3029sub1_objecttype = 7
  p3029sub1_datatype = 6
  p3029sub1_lowlimit = 
  p3029sub1_highlimit = 
  p3029sub1_accesstype = rw
  p3029sub1_pdomapping = 0
  p3029sub1_parametervalue = 
  p3029sub1_objflags = 0
  p3029sub2_parametername = Manual.stateMan
  p3029sub2_objecttype = 7
  p3029sub2_datatype = 6
  p3029sub2_lowlimit = 
  p3029sub2_highlimit = 
  p3029sub2_accesstype = ro
  p3029sub2_pdomapping = 0
  p3029sub4_parametername = Manual.n_slowMan
  p3029sub4_objecttype = 7
  p3029sub4_datatype = 6
  p3029sub4_accesstype = rw
  p3029sub4_pdomapping = 0
  p3029sub4_parametervalue = 
  p3029sub4_objflags = 0
  p3029sub5_parametername = Manual.n_fastMan
  p3029sub5_objecttype = 7
  p3029sub5_datatype = 6
  p3029sub5_accesstype = rw
  p3029sub5_pdomapping = 0
  p3029sub5_parametervalue = 
  p3029sub5_objflags = 0
  p3029sub7_parametername = Manual.step_Man
  p3029sub7_objecttype = 7
  p3029sub7_datatype = 6
  p3029sub7_lowlimit = 
  p3029sub7_highlimit = 
  p3029sub7_accesstype = rw
  p3029sub7_pdomapping = 0
  p3029sub7_parametervalue = 
  p3029sub7_objflags = 0
  p3029sub8_parametername = Manual.time_Man
  p3029sub8_objecttype = 7
  p3029sub8_datatype = 6
  p3029sub8_lowlimit = 
  p3029sub8_highlimit = 
  p3029sub8_accesstype = rw
  p3029sub8_pdomapping = 0
  p3029sub8_parametervalue = 
  p3029sub8_objflags = 0
  p3320_parametername = prog io0
  p3320_objecttype = 9
  p3320_subnumber = 0x7
  p3320_parametervalue = 
  p3320_objflags = 0
  p3320sub0_parametername = number of entries
  p3320sub0_objecttype = 7
  p3320sub0_datatype = 5
  p3320sub0_accesstype = ro
  p3320sub0_pdomapping = 0
  p3320sub1_parametername = ProgIO0.Index
  p3320sub1_objecttype = 7
  p3320sub1_datatype = 6
  p3320sub1_lowlimit = 
  p3320sub1_highlimit = 
  p3320sub1_accesstype = rw
  p3320sub1_pdomapping = 0
  p3320sub1_parametervalue = 
  p3320sub1_objflags = 0
  p3320sub2_parametername = ProgIO0.Subindex
  p3320sub2_objecttype = 7
  p3320sub2_datatype = 6
  p3320sub2_lowlimit = 
  p3320sub2_highlimit = 
  p3320sub2_accesstype = rw
  p3320sub2_pdomapping = 0
  p3320sub2_parametervalue = 
  p3320sub2_objflags = 0
  p3320sub3_parametername = ProgIO0.BitMask
  p3320sub3_objecttype = 7
  p3320sub3_datatype = 7
  p3320sub3_lowlimit = 
  p3320sub3_highlimit = 
  p3320sub3_accesstype = rw
  p3320sub3_pdomapping = 0
  p3320sub3_parametervalue = 
  p3320sub3_objflags = 0
  p3320sub4_parametername = ProgIO0.Switch
  p3320sub4_objecttype = 7
  p3320sub4_datatype = 6
  p3320sub4_lowlimit = 
  p3320sub4_highlimit = 
  p3320sub4_accesstype = rw
  p3320sub4_pdomapping = 0
  p3320sub4_parametervalue = 
  p3320sub4_objflags = 0
  p3320sub5_parametername = ProgIO0.Value1
  p3320sub5_objecttype = 7
  p3320sub5_datatype = 4
  p3320sub5_lowlimit = 
  p3320sub5_highlimit = 
  p3320sub5_accesstype = rw
  p3320sub5_pdomapping = 0
  p3320sub5_parametervalue = 
  p3320sub5_objflags = 0
  p3320sub6_parametername = ProgIO0.Value2
  p3320sub6_objecttype = 7
  p3320sub6_datatype = 4
  p3320sub6_lowlimit = 
  p3320sub6_highlimit = 
  p3320sub6_accesstype = rw
  p3320sub6_pdomapping = 0
  p3320sub6_parametervalue = 
  p3320sub6_objflags = 0
  p3321_parametername = prog io1
  p3321_objecttype = 9
  p3321_subnumber = 0x7
  p3321_parametervalue = 
  p3321_objflags = 0
  p3321sub0_parametername = number of entries
  p3321sub0_objecttype = 7
  p3321sub0_datatype = 5
  p3321sub0_accesstype = ro
  p3321sub0_pdomapping = 0
  p3321sub1_parametername = ProgIO1.Index
  p3321sub1_objecttype = 7
  p3321sub1_datatype = 6
  p3321sub1_lowlimit = 
  p3321sub1_highlimit = 
  p3321sub1_accesstype = rw
  p3321sub1_pdomapping = 0
  p3321sub1_parametervalue = 
  p3321sub1_objflags = 0
  p3321sub2_parametername = ProgIO1.Subindex
  p3321sub2_objecttype = 7
  p3321sub2_datatype = 6
  p3321sub2_lowlimit = 
  p3321sub2_highlimit = 
  p3321sub2_accesstype = rw
  p3321sub2_pdomapping = 0
  p3321sub2_parametervalue = 
  p3321sub2_objflags = 0
  p3321sub3_parametername = ProgIO1.BitMask
  p3321sub3_objecttype = 7
  p3321sub3_datatype = 7
  p3321sub3_lowlimit = 
  p3321sub3_highlimit = 
  p3321sub3_accesstype = rw
  p3321sub3_pdomapping = 0
  p3321sub3_parametervalue = 
  p3321sub3_objflags = 0
  p3321sub4_parametername = ProgIO1.Switch
  p3321sub4_objecttype = 7
  p3321sub4_datatype = 6
  p3321sub4_lowlimit = 
  p3321sub4_highlimit = 
  p3321sub4_accesstype = rw
  p3321sub4_pdomapping = 0
  p3321sub4_parametervalue = 
  p3321sub4_objflags = 0
  p3321sub5_parametername = ProgIO1.Value1
  p3321sub5_objecttype = 7
  p3321sub5_datatype = 4
  p3321sub5_lowlimit = 
  p3321sub5_highlimit = 
  p3321sub5_accesstype = rw
  p3321sub5_pdomapping = 0
  p3321sub5_parametervalue = 
  p3321sub5_objflags = 0
  p3321sub6_parametername = ProgIO1.Value2
  p3321sub6_objecttype = 7
  p3321sub6_datatype = 4
  p3321sub6_lowlimit = 
  p3321sub6_highlimit = 
  p3321sub6_accesstype = rw
  p3321sub6_pdomapping = 0
  p3321sub6_parametervalue = 
  p3321sub6_objflags = 0
  p3322_parametername = prog io2
  p3322_objecttype = 9
  p3322_subnumber = 0x7
  p3322_parametervalue = 
  p3322_objflags = 0
  p3322sub0_parametername = number of entries
  p3322sub0_objecttype = 7
  p3322sub0_datatype = 5
  p3322sub0_accesstype = ro
  p3322sub0_pdomapping = 0
  p3322sub1_parametername = ProgIO2.Index
  p3322sub1_objecttype = 7
  p3322sub1_datatype = 6
  p3322sub1_lowlimit = 
  p3322sub1_highlimit = 
  p3322sub1_accesstype = rw
  p3322sub1_pdomapping = 0
  p3322sub1_parametervalue = 
  p3322sub1_objflags = 0
  p3322sub2_parametername = ProgIO2.Subindex
  p3322sub2_objecttype = 7
  p3322sub2_datatype = 6
  p3322sub2_lowlimit = 
  p3322sub2_highlimit = 
  p3322sub2_accesstype = rw
  p3322sub2_pdomapping = 0
  p3322sub2_parametervalue = 
  p3322sub2_objflags = 0
  p3322sub3_parametername = ProgIO2.BitMask
  p3322sub3_objecttype = 7
  p3322sub3_datatype = 7
  p3322sub3_lowlimit = 
  p3322sub3_highlimit = 
  p3322sub3_accesstype = rw
  p3322sub3_pdomapping = 0
  p3322sub3_parametervalue = 
  p3322sub3_objflags = 0
  p3322sub4_parametername = ProgIO2.Switch
  p3322sub4_objecttype = 7
  p3322sub4_datatype = 6
  p3322sub4_lowlimit = 
  p3322sub4_highlimit = 
  p3322sub4_accesstype = rw
  p3322sub4_pdomapping = 0
  p3322sub4_parametervalue = 
  p3322sub4_objflags = 0
  p3322sub5_parametername = ProgIO2.Value1
  p3322sub5_objecttype = 7
  p3322sub5_datatype = 4
  p3322sub5_lowlimit = 
  p3322sub5_highlimit = 
  p3322sub5_accesstype = rw
  p3322sub5_pdomapping = 0
  p3322sub5_parametervalue = 
  p3322sub5_objflags = 0
  p3322sub6_parametername = ProgIO2.Value2
  p3322sub6_objecttype = 7
  p3322sub6_datatype = 4
  p3322sub6_lowlimit = 
  p3322sub6_highlimit = 
  p3322sub6_accesstype = rw
  p3322sub6_pdomapping = 0
  p3322sub6_parametervalue = 
  p3322sub6_objflags = 0
  p3323_parametername = prog io3
  p3323_objecttype = 9
  p3323_subnumber = 0x7
  p3323_parametervalue = 
  p3323_objflags = 0
  p3323sub0_parametername = number of entries
  p3323sub0_objecttype = 7
  p3323sub0_datatype = 5
  p3323sub0_accesstype = ro
  p3323sub0_pdomapping = 0
  p3323sub1_parametername = ProgIO3.Index
  p3323sub1_objecttype = 7
  p3323sub1_datatype = 6
  p3323sub1_lowlimit = 
  p3323sub1_highlimit = 
  p3323sub1_accesstype = rw
  p3323sub1_pdomapping = 0
  p3323sub1_parametervalue = 
  p3323sub1_objflags = 0
  p3323sub2_parametername = ProgIO3.Subindex
  p3323sub2_objecttype = 7
  p3323sub2_datatype = 6
  p3323sub2_lowlimit = 
  p3323sub2_highlimit = 
  p3323sub2_accesstype = rw
  p3323sub2_pdomapping = 0
  p3323sub2_parametervalue = 
  p3323sub2_objflags = 0
  p3323sub3_parametername = ProgIO3.BitMask
  p3323sub3_objecttype = 7
  p3323sub3_datatype = 7
  p3323sub3_lowlimit = 
  p3323sub3_highlimit = 
  p3323sub3_accesstype = rw
  p3323sub3_pdomapping = 0
  p3323sub3_parametervalue = 
  p3323sub3_objflags = 0
  p3323sub4_parametername = ProgIO3.Switch
  p3323sub4_objecttype = 7
  p3323sub4_datatype = 6
  p3323sub4_lowlimit = 
  p3323sub4_highlimit = 
  p3323sub4_accesstype = rw
  p3323sub4_pdomapping = 0
  p3323sub4_parametervalue = 
  p3323sub4_objflags = 0
  p3323sub5_parametername = ProgIO3.Value1
  p3323sub5_objecttype = 7
  p3323sub5_datatype = 4
  p3323sub5_lowlimit = 
  p3323sub5_highlimit = 
  p3323sub5_accesstype = rw
  p3323sub5_pdomapping = 0
  p3323sub5_parametervalue = 
  p3323sub5_objflags = 0
  p3323sub6_parametername = ProgIO3.Value2
  p3323sub6_objecttype = 7
  p3323sub6_datatype = 4
  p3323sub6_lowlimit = 
  p3323sub6_highlimit = 
  p3323sub6_accesstype = rw
  p3323sub6_pdomapping = 0
  p3323sub6_parametervalue = 
  p3323sub6_objflags = 0
ILE1F_BK2 : FBC.0x0100002E.1.SEILE1F_0110E v1.10 (OrderNumber=ILE1F)  [CAN1 -> SI_unit_BK1.CAN2 (NodeNumber=7)]
  p1403_transmissionselection = 1
  plifeguarding_guardtime = 500
  plifeguarding_retryfactor = 10
  p3001_parametername = mandatory
  p3001_objecttype = 9
  p3001_subnumber = 0x3
  p3001_parametervalue = 
  p3001_objflags = 0
  p3001sub0_parametername = number of entries
  p3001sub0_objecttype = 7
  p3001sub0_datatype = 5
  p3001sub0_accesstype = ro
  p3001sub0_pdomapping = 0
  p3001sub1_parametername = Config.PrgNo
  p3001sub1_objecttype = 7
  p3001sub1_datatype = 7
  p3001sub1_lowlimit = 
  p3001sub1_highlimit = 
  p3001sub1_accesstype = ro
  p3001sub1_pdomapping = 0
  p3001sub2_parametername = Config.PrgVer
  p3001sub2_objecttype = 7
  p3001sub2_datatype = 7
  p3001sub2_lowlimit = 
  p3001sub2_highlimit = 
  p3001sub2_accesstype = ro
  p3001sub2_pdomapping = 0
  p300b_parametername = system settings
  p300b_objecttype = 9
  p300b_subnumber = 0x7
  p300b_parametervalue = 
  p300b_objflags = 0
  p300bsub0_parametername = number of entries
  p300bsub0_objecttype = 7
  p300bsub0_datatype = 5
  p300bsub0_accesstype = ro
  p300bsub0_pdomapping = 0
  p300bsub1_parametername = Settings.name1
  p300bsub1_objecttype = 7
  p300bsub1_datatype = 7
  p300bsub1_lowlimit = 
  p300bsub1_highlimit = 
  p300bsub1_accesstype = rw
  p300bsub1_pdomapping = 0
  p300bsub1_parametervalue = 
  p300bsub1_objflags = 0
  p300bsub2_parametername = Settings.name2
  p300bsub2_objecttype = 7
  p300bsub2_datatype = 7
  p300bsub2_lowlimit = 
  p300bsub2_highlimit = 
  p300bsub2_accesstype = rw
  p300bsub2_pdomapping = 0
  p300bsub2_parametervalue = 
  p300bsub2_objflags = 0
  p300bsub6_parametername = Commands.eeprSave
  p300bsub6_objecttype = 7
  p300bsub6_datatype = 6
  p300bsub6_lowlimit = 
  p300bsub6_highlimit = 
  p300bsub6_accesstype = rw
  p300bsub6_pdomapping = 0
  p300bsub6_parametervalue = 1
  p300bsub6_objflags = 0
  p300bsub7_parametername = Commands.stateSave
  p300bsub7_objecttype = 7
  p300bsub7_datatype = 6
  p300bsub7_lowlimit = 
  p300bsub7_highlimit = 
  p300bsub7_accesstype = ro
  p300bsub7_pdomapping = 0
  p300bsub8_parametername = Commands.default
  p300bsub8_objecttype = 7
  p300bsub8_datatype = 6
  p300bsub8_lowlimit = 
  p300bsub8_highlimit = 
  p300bsub8_accesstype = rw
  p300bsub8_pdomapping = 0
  p300bsub8_parametervalue = 
  p300bsub8_objflags = 0
  p300bsub9_parametername = Commands.stateDef
  p300bsub9_objecttype = 7
  p300bsub9_datatype = 6
  p300bsub9_lowlimit = 
  p300bsub9_highlimit = 
  p300bsub9_accesstype = ro
  p300bsub9_pdomapping = 0
  p300f_parametername = controller  settings
  p300f_objecttype = 9
  p300f_subnumber = 0xE
  p300f_parametervalue = 
  p300f_objflags = 0
  p300fsub0_parametername = number of entries
  p300fsub0_objecttype = 7
  p300fsub0_datatype = 5
  p300fsub0_accesstype = ro
  p300fsub0_pdomapping = 0
  p300fsub1_parametername = Config.I_nomDrv
  p300fsub1_objecttype = 7
  p300fsub1_datatype = 6
  p300fsub1_accesstype = ro
  p300fsub1_pdomapping = 0
  p300fsub2_parametername = Config.I_maxDrv
  p300fsub2_objecttype = 7
  p300fsub2_datatype = 6
  p300fsub2_accesstype = ro
  p300fsub2_pdomapping = 0
  p300fsub3_parametername = Settings.I_max
  p300fsub3_objecttype = 7
  p300fsub3_datatype = 6
  p300fsub3_accesstype = rw
  p300fsub3_pdomapping = 0
  p300fsub3_parametervalue = 60
  p300fsub3_objflags = 0
  p300fsub5_parametername = Settings.I_maxBlk
  p300fsub5_objecttype = 7
  p300fsub5_datatype = 6
  p300fsub5_lowlimit = 
  p300fsub5_highlimit = 
  p300fsub5_accesstype = rw
  p300fsub5_pdomapping = 0
  p300fsub5_parametervalue = 20
  p300fsub5_objflags = 0
  p300fsub7_parametername = Settings.p_maxDiff
  p300fsub7_objecttype = 7
  p300fsub7_datatype = 6
  p300fsub7_lowlimit = 
  p300fsub7_highlimit = 
  p300fsub7_accesstype = rw
  p300fsub7_pdomapping = 0
  p300fsub7_parametervalue = 24
  p300fsub7_objflags = 0
  p300fsub8_parametername = Control.KPn
  p300fsub8_objecttype = 7
  p300fsub8_datatype = 6
  p300fsub8_lowlimit = 
  p300fsub8_highlimit = 
  p300fsub8_accesstype = rw
  p300fsub8_pdomapping = 0
  p300fsub8_parametervalue = 60
  p300fsub8_objflags = 0
  p300fsub9_parametername = Control.TNn
  p300fsub9_objecttype = 7
  p300fsub9_datatype = 6
  p300fsub9_lowlimit = 
  p300fsub9_highlimit = 
  p300fsub9_accesstype = rw
  p300fsub9_pdomapping = 0
  p300fsub9_parametervalue = 10000
  p300fsub9_objflags = 0
  p300fsuba_parametername = Control.KPp
  p300fsuba_objecttype = 7
  p300fsuba_datatype = 6
  p300fsuba_lowlimit = 
  p300fsuba_highlimit = 
  p300fsuba_accesstype = rw
  p300fsuba_pdomapping = 0
  p300fsuba_parametervalue = 300
  p300fsuba_objflags = 0
  p300fsubb_parametername = Control.KFPp
  p300fsubb_objecttype = 7
  p300fsubb_datatype = 6
  p300fsubb_lowlimit = 
  p300fsubb_highlimit = 
  p300fsubb_accesstype = rw
  p300fsubb_pdomapping = 0
  p300fsubb_parametervalue = 32767
  p300fsubb_objflags = 0
  p300fsubc_parametername = Settings.T_block
  p300fsubc_objecttype = 7
  p300fsubc_datatype = 6
  p300fsubc_lowlimit = 
  p300fsubc_highlimit = 
  p300fsubc_accesstype = rw
  p300fsubc_pdomapping = 0
  p300fsubc_parametervalue = 100
  p300fsubc_objflags = 0
  p300fsubd_parametername = Status.p_difPeak
  p300fsubd_objecttype = 7
  p300fsubd_datatype = 7
  p300fsubd_lowlimit = 
  p300fsubd_highlimit = 
  p300fsubd_accesstype = rw
  p300fsubd_pdomapping = 0
  p300fsubd_parametervalue = 
  p300fsubd_objflags = 0
  p300fsubf_parametername = Settings.p_win
  p300fsubf_objecttype = 7
  p300fsubf_datatype = 6
  p300fsubf_lowlimit = 
  p300fsubf_highlimit = 
  p300fsubf_accesstype = rw
  p300fsubf_pdomapping = 0
  p300fsubf_parametervalue = 1
  p300fsubf_objflags = 0
  p300fsub10_parametername = Settings.p_winTime
  p300fsub10_objecttype = 7
  p300fsub10_datatype = 6
  p300fsub10_lowlimit = 
  p300fsub10_highlimit = 
  p300fsub10_accesstype = rw
  p300fsub10_pdomapping = 0
  p300fsub10_parametervalue = 0
  p300fsub10_objflags = 0
  p3016_parametername = rs485
  p3016_objecttype = 9
  p3016_subnumber = 0x4
  p3016_parametervalue = 
  p3016_objflags = 0
  p3016sub0_parametername = number of entries
  p3016sub0_objecttype = 7
  p3016sub0_datatype = 5
  p3016sub0_accesstype = ro
  p3016sub0_pdomapping = 0
  p3016sub1_parametername = RS485.serBaud
  p3016sub1_objecttype = 7
  p3016sub1_datatype = 6
  p3016sub1_lowlimit = 
  p3016sub1_highlimit = 
  p3016sub1_accesstype = rw
  p3016sub1_pdomapping = 0
  p3016sub1_parametervalue = 
  p3016sub1_objflags = 0
  p3016sub2_parametername = RS485.serAdr
  p3016sub2_objecttype = 7
  p3016sub2_datatype = 6
  p3016sub2_lowlimit = 
  p3016sub2_highlimit = 
  p3016sub2_accesstype = rw
  p3016sub2_pdomapping = 0
  p3016sub2_parametervalue = 
  p3016sub2_objflags = 0
  p3016sub3_parametername = RS485.serFormat
  p3016sub3_objecttype = 7
  p3016sub3_datatype = 6
  p3016sub3_lowlimit = 
  p3016sub3_highlimit = 
  p3016sub3_accesstype = rw
  p3016sub3_pdomapping = 0
  p3016sub3_parametervalue = 
  p3016sub3_objflags = 0
  p3017_parametername = can
  p3017_objecttype = 9
  p3017_subnumber = 0x3
  p3017_parametervalue = 
  p3017_objflags = 0
  p3017sub0_parametername = number of entries
  p3017sub0_objecttype = 7
  p3017sub0_datatype = 5
  p3017sub0_accesstype = ro
  p3017sub0_pdomapping = 0
  p3017sub2_parametername = CAN.canAddr
  p3017sub2_objecttype = 7
  p3017sub2_datatype = 6
  p3017sub2_lowlimit = 
  p3017sub2_highlimit = 
  p3017sub2_accesstype = rw
  p3017sub2_pdomapping = 0
  p3017sub2_parametervalue = 
  p3017sub2_objflags = 0
  p3017sub3_parametername = CAN.canBaud
  p3017sub3_objecttype = 7
  p3017sub3_datatype = 6
  p3017sub3_lowlimit = 
  p3017sub3_highlimit = 
  p3017sub3_accesstype = rw
  p3017sub3_pdomapping = 0
  p3017sub3_parametervalue = 
  p3017sub3_objflags = 0
  p301c_parametername = settings1
  p301c_objecttype = 9
  p301c_subnumber = 0xF
  p301c_parametervalue = 
  p301c_objflags = 0
  p301csub0_parametername = number of entries
  p301csub0_objecttype = 7
  p301csub0_datatype = 5
  p301csub0_accesstype = ro
  p301csub0_pdomapping = 0
  p301csub3_parametername = Status.xMode_act
  p301csub3_objecttype = 7
  p301csub3_datatype = 6
  p301csub3_lowlimit = 
  p301csub3_highlimit = 
  p301csub3_accesstype = ro
  p301csub3_pdomapping = 0
  p301csub6_parametername = Motion.invertDir
  p301csub6_objecttype = 7
  p301csub6_datatype = 6
  p301csub6_lowlimit = 
  p301csub6_highlimit = 
  p301csub6_accesstype = rw
  p301csub6_pdomapping = 0
  p301csub6_parametervalue = 0
  p301csub6_objflags = 0
  p301csuba_parametername = Status.WarnSig
  p301csuba_objecttype = 7
  p301csuba_datatype = 6
  p301csuba_lowlimit = 
  p301csuba_highlimit = 
  p301csuba_accesstype = ro
  p301csuba_pdomapping = 0
  p301csubb_parametername = Settings.WarnOvrun
  p301csubb_objecttype = 7
  p301csubb_datatype = 6
  p301csubb_lowlimit = 
  p301csubb_highlimit = 
  p301csubb_accesstype = rw
  p301csubb_pdomapping = 0
  p301csubb_parametervalue = 0
  p301csubb_objflags = 0
  p301csubd_parametername = Settings.SignEnabl
  p301csubd_objecttype = 7
  p301csubd_datatype = 6
  p301csubd_lowlimit = 
  p301csubd_highlimit = 
  p301csubd_accesstype = rw
  p301csubd_pdomapping = 0
  p301csubd_parametervalue = 3
  p301csubd_objflags = 0
  p301csube_parametername = Settings.SignLevel
  p301csube_objecttype = 7
  p301csube_datatype = 6
  p301csube_lowlimit = 
  p301csube_highlimit = 
  p301csube_accesstype = rw
  p301csube_pdomapping = 0
  p301csube_parametervalue = 0
  p301csube_objflags = 0
  p301csubf_parametername = Status.Sign_SR
  p301csubf_objecttype = 7
  p301csubf_datatype = 6
  p301csubf_lowlimit = 
  p301csubf_highlimit = 
  p301csubf_accesstype = ro
  p301csubf_pdomapping = 0
  p301csub11_parametername = Status.FltSig
  p301csub11_objecttype = 7
  p301csub11_datatype = 7
  p301csub11_lowlimit = 
  p301csub11_highlimit = 
  p301csub11_accesstype = ro
  p301csub11_pdomapping = 0
  p301csub12_parametername = Status.FltSig_SR
  p301csub12_objecttype = 7
  p301csub12_datatype = 7
  p301csub12_lowlimit = 
  p301csub12_highlimit = 
  p301csub12_accesstype = ro
  p301csub12_pdomapping = 0
  p301csub13_parametername = Status.action_st
  p301csub13_objecttype = 7
  p301csub13_datatype = 6
  p301csub13_lowlimit = 
  p301csub13_highlimit = 
  p301csub13_accesstype = ro
  p301csub13_pdomapping = 0
  p301csub15_parametername = Motion.dec_Stop
  p301csub15_objecttype = 7
  p301csub15_datatype = 7
  p301csub15_lowlimit = 
  p301csub15_highlimit = 
  p301csub15_accesstype = rw
  p301csub15_pdomapping = 0
  p301csub15_parametervalue = 4960
  p301csub15_objflags = 0
  p301csub18_parametername = Settings.Flt_pDiff
  p301csub18_objecttype = 7
  p301csub18_datatype = 6
  p301csub18_lowlimit = 
  p301csub18_highlimit = 
  p301csub18_accesstype = rw
  p301csub18_pdomapping = 0
  p301csub18_parametervalue = 3
  p301csub18_objflags = 0
  p301d_parametername = settings2
  p301d_objecttype = 9
  p301d_subnumber = 0x4
  p301d_parametervalue = 
  p301d_objflags = 0
  p301dsub0_parametername = number of entries
  p301dsub0_objecttype = 7
  p301dsub0_datatype = 5
  p301dsub0_accesstype = ro
  p301dsub0_pdomapping = 0
  p301dsub2_parametername = Config.ResolutM
  p301dsub2_objecttype = 7
  p301dsub2_datatype = 6
  p301dsub2_accesstype = ro
  p301dsub2_pdomapping = 0
  p301dsub17_parametername = Motion.v_target0
  p301dsub17_objecttype = 7
  p301dsub17_datatype = 6
  p301dsub17_accesstype = rw
  p301dsub17_pdomapping = 0
  p301dsub17_parametervalue = 1000
  p301dsub17_objflags = 0
  p301dsub1a_parametername = Motion.acc
  p301dsub1a_objecttype = 7
  p301dsub1a_datatype = 7
  p301dsub1a_lowlimit = 
  p301dsub1a_highlimit = 
  p301dsub1a_accesstype = rw
  p301dsub1a_pdomapping = 0
  p301dsub1a_parametervalue = 2442
  p301dsub1a_objflags = 0
  p301e_parametername = pdo data
  p301e_objecttype = 9
  p301e_subnumber = 0xC
  p301e_parametervalue = 
  p301e_objflags = 0
  p301esub0_parametername = number of entries
  p301esub0_objecttype = 7
  p301esub0_datatype = 5
  p301esub0_accesstype = ro
  p301esub0_pdomapping = 0
  p301esubb_parametername = Status.ModeError
  p301esubb_objecttype = 7
  p301esubb_datatype = 6
  p301esubb_lowlimit = 
  p301esubb_highlimit = 
  p301esubb_accesstype = ro
  p301esubb_pdomapping = 0
  p301f_parametername = status
  p301f_objecttype = 9
  p301f_subnumber = 0x11
  p301f_parametervalue = 
  p301f_objflags = 0
  p301fsub0_parametername = number of entries
  p301fsub0_objecttype = 7
  p301fsub0_datatype = 5
  p301fsub0_accesstype = ro
  p301fsub0_pdomapping = 0
  p301fsub1_parametername = Status.v_ref
  p301fsub1_objecttype = 7
  p301fsub1_datatype = 4
  p301fsub1_lowlimit = 
  p301fsub1_highlimit = 
  p301fsub1_accesstype = ro
  p301fsub1_pdomapping = 0
  p301fsub2_parametername = Status.v_act
  p301fsub2_objecttype = 7
  p301fsub2_datatype = 4
  p301fsub2_lowlimit = 
  p301fsub2_highlimit = 
  p301fsub2_accesstype = ro
  p301fsub2_pdomapping = 0
  p301fsub5_parametername = Status.p_ref
  p301fsub5_objecttype = 7
  p301fsub5_datatype = 4
  p301fsub5_lowlimit = 
  p301fsub5_highlimit = 
  p301fsub5_accesstype = ro
  p301fsub5_pdomapping = 0
  p301fsub6_parametername = Status.p_act
  p301fsub6_objecttype = 7
  p301fsub6_datatype = 4
  p301fsub6_lowlimit = 
  p301fsub6_highlimit = 
  p301fsub6_accesstype = ro
  p301fsub6_pdomapping = 0
  p301fsub7_parametername = Status.p_dif
  p301fsub7_objecttype = 7
  p301fsub7_datatype = 4
  p301fsub7_lowlimit = 
  p301fsub7_highlimit = 
  p301fsub7_accesstype = ro
  p301fsub7_pdomapping = 0
  p301fsub8_parametername = Status.n_ref
  p301fsub8_objecttype = 7
  p301fsub8_datatype = 3
  p301fsub8_lowlimit = 
  p301fsub8_highlimit = 
  p301fsub8_accesstype = ro
  p301fsub8_pdomapping = 0
  p301fsub9_parametername = Status.n_act
  p301fsub9_objecttype = 7
  p301fsub9_datatype = 3
  p301fsub9_lowlimit = 
  p301fsub9_highlimit = 
  p301fsub9_accesstype = ro
  p301fsub9_pdomapping = 0
  p301fsubc_parametername = Status.I_act
  p301fsubc_objecttype = 7
  p301fsubc_datatype = 3
  p301fsubc_lowlimit = 
  p301fsubc_highlimit = 
  p301fsubc_accesstype = ro
  p301fsubc_pdomapping = 0
  p301fsub14_parametername = Status.UDC_act
  p301fsub14_objecttype = 7
  p301fsub14_datatype = 6
  p301fsub14_lowlimit = 
  p301fsub14_highlimit = 
  p301fsub14_accesstype = ro
  p301fsub14_pdomapping = 0
  p301fsub19_parametername = Status.TPA_act
  p301fsub19_objecttype = 7
  p301fsub19_datatype = 6
  p301fsub19_lowlimit = 
  p301fsub19_highlimit = 
  p301fsub19_accesstype = ro
  p301fsub19_pdomapping = 0
  p301fsub1c_parametername = Status.v_pref
  p301fsub1c_objecttype = 7
  p301fsub1c_datatype = 4
  p301fsub1c_lowlimit = 
  p301fsub1c_highlimit = 
  p301fsub1c_accesstype = ro
  p301fsub1c_pdomapping = 0
  p301fsub1e_parametername = Status.p_target
  p301fsub1e_objecttype = 7
  p301fsub1e_datatype = 4
  p301fsub1e_lowlimit = 
  p301fsub1e_highlimit = 
  p301fsub1e_accesstype = ro
  p301fsub1e_pdomapping = 0
  p301fsub1f_parametername = Status.p_profile
  p301fsub1f_objecttype = 7
  p301fsub1f_datatype = 4
  p301fsub1f_lowlimit = 
  p301fsub1f_highlimit = 
  p301fsub1f_accesstype = ro
  p301fsub1f_pdomapping = 0
  p301fsub23_parametername = Status.n_profile
  p301fsub23_objecttype = 7
  p301fsub23_datatype = 3
  p301fsub23_lowlimit = 
  p301fsub23_highlimit = 
  p301fsub23_accesstype = ro
  p301fsub23_pdomapping = 0
  p301fsub26_parametername = Status.n_target
  p301fsub26_objecttype = 7
  p301fsub26_datatype = 3
  p301fsub26_lowlimit = 
  p301fsub26_highlimit = 
  p301fsub26_accesstype = ro
  p301fsub26_pdomapping = 0
  p301fsub2d_parametername = Status.n_pref
  p301fsub2d_objecttype = 7
  p301fsub2d_datatype = 3
  p301fsub2d_lowlimit = 
  p301fsub2d_highlimit = 
  p301fsub2d_accesstype = ro
  p301fsub2d_pdomapping = 0
  p3020_parametername = error
  p3020_objecttype = 9
  p3020_subnumber = 0x5
  p3020_parametervalue = 
  p3020_objflags = 0
  p3020sub0_parametername = number of entries
  p3020sub0_objecttype = 7
  p3020sub0_datatype = 5
  p3020sub0_accesstype = ro
  p3020sub0_pdomapping = 0
  p3020sub1_parametername = ErrorMemAvailable
  p3020sub1_objecttype = 7
  p3020sub1_datatype = 6
  p3020sub1_lowlimit = 
  p3020sub1_highlimit = 
  p3020sub1_accesstype = ro
  p3020sub1_pdomapping = 0
  p3020sub2_parametername = Commands.del_err
  p3020sub2_objecttype = 7
  p3020sub2_datatype = 6
  p3020sub2_lowlimit = 
  p3020sub2_highlimit = 
  p3020sub2_accesstype = rw
  p3020sub2_pdomapping = 0
  p3020sub2_parametervalue = 
  p3020sub2_objflags = 0
  p3020sub6_parametername = PowerOnCount
  p3020sub6_objecttype = 7
  p3020sub6_datatype = 7
  p3020sub6_lowlimit = 
  p3020sub6_highlimit = 
  p3020sub6_accesstype = ro
  p3020sub6_pdomapping = 0
  p3020sub7_parametername = Status.StopFault
  p3020sub7_objecttype = 7
  p3020sub7_datatype = 6
  p3020sub7_lowlimit = 
  p3020sub7_highlimit = 
  p3020sub7_accesstype = ro
  p3020sub7_pdomapping = 0
  p3021_parametername = io
  p3021_objecttype = 9
  p3021_subnumber = 0x4
  p3021_parametervalue = 
  p3021_objflags = 0
  p3021sub0_parametername = number of entries
  p3021sub0_objecttype = 7
  p3021sub0_datatype = 5
  p3021sub0_accesstype = ro
  p3021sub0_pdomapping = 0
  p3021sub1_parametername = I/O.IO_act
  p3021sub1_objecttype = 7
  p3021sub1_datatype = 6
  p3021sub1_lowlimit = 
  p3021sub1_highlimit = 
  p3021sub1_accesstype = rw
  p3021sub1_pdomapping = 0
  p3021sub1_parametervalue = 
  p3021sub1_objflags = 0
  p3021sub7_parametername = Commands.brake
  p3021sub7_objecttype = 7
  p3021sub7_datatype = 6
  p3021sub7_lowlimit = 
  p3021sub7_highlimit = 
  p3021sub7_accesstype = rw
  p3021sub7_pdomapping = 0
  p3021sub7_parametervalue = 
  p3021sub7_objflags = 0
  p3021sub8_parametername = Status.brake
  p3021sub8_objecttype = 7
  p3021sub8_datatype = 6
  p3021sub8_lowlimit = 
  p3021sub8_highlimit = 
  p3021sub8_accesstype = ro
  p3021sub8_pdomapping = 0
  p3022_parametername = io definitions
  p3022_objecttype = 9
  p3022_subnumber = 0x6
  p3022_parametervalue = 
  p3022_objflags = 0
  p3022sub0_parametername = number of entries
  p3022sub0_objecttype = 7
  p3022sub0_datatype = 5
  p3022sub0_accesstype = ro
  p3022sub0_pdomapping = 0
  p3022sub1_parametername = I/O.IO0_def
  p3022sub1_objecttype = 7
  p3022sub1_datatype = 6
  p3022sub1_lowlimit = 
  p3022sub1_highlimit = 
  p3022sub1_accesstype = rw
  p3022sub1_pdomapping = 0
  p3022sub1_parametervalue = 0
  p3022sub1_objflags = 0
  p3022sub2_parametername = I/O.IO1_def
  p3022sub2_objecttype = 7
  p3022sub2_datatype = 6
  p3022sub2_lowlimit = 
  p3022sub2_highlimit = 
  p3022sub2_accesstype = rw
  p3022sub2_pdomapping = 0
  p3022sub2_parametervalue = 0
  p3022sub2_objflags = 0
  p3022sub3_parametername = I/O.IO2_def
  p3022sub3_objecttype = 7
  p3022sub3_datatype = 6
  p3022sub3_lowlimit = 
  p3022sub3_highlimit = 
  p3022sub3_accesstype = rw
  p3022sub3_pdomapping = 0
  p3022sub3_parametervalue = 0
  p3022sub3_objflags = 0
  p3022sub4_parametername = I/O.IO3_def
  p3022sub4_objecttype = 7
  p3022sub4_datatype = 6
  p3022sub4_lowlimit = 
  p3022sub4_highlimit = 
  p3022sub4_accesstype = rw
  p3022sub4_pdomapping = 0
  p3022sub4_parametervalue = 
  p3022sub4_objflags = 0
  p3022sub7_parametername = I/O.progDelay
  p3022sub7_objecttype = 7
  p3022sub7_datatype = 6
  p3022sub7_lowlimit = 
  p3022sub7_highlimit = 
  p3022sub7_accesstype = rw
  p3022sub7_pdomapping = 0
  p3022sub7_parametervalue = 
  p3022sub7_objflags = 0
  p3023_parametername = ptp
  p3023_objecttype = 9
  p3023_subnumber = 0x6
  p3023_parametervalue = 
  p3023_objflags = 0
  p3023sub0_parametername = number of entries
  p3023sub0_objecttype = 7
  p3023sub0_datatype = 5
  p3023sub0_accesstype = ro
  p3023sub0_pdomapping = 0
  p3023sub1_parametername = PTP.p_absPTP
  p3023sub1_objecttype = 7
  p3023sub1_datatype = 4
  p3023sub1_lowlimit = 
  p3023sub1_highlimit = 
  p3023sub1_accesstype = rw
  p3023sub1_pdomapping = 0
  p3023sub1_parametervalue = 
  p3023sub1_objflags = 0
  p3023sub2_parametername = PTP.StatePTP
  p3023sub2_objecttype = 7
  p3023sub2_datatype = 6
  p3023sub2_lowlimit = 
  p3023sub2_highlimit = 
  p3023sub2_accesstype = ro
  p3023sub2_pdomapping = 0
  p3023sub3_parametername = PTP.p_relPTP
  p3023sub3_objecttype = 7
  p3023sub3_datatype = 4
  p3023sub3_lowlimit = 
  p3023sub3_highlimit = 
  p3023sub3_accesstype = rw
  p3023sub3_pdomapping = 0
  p3023sub3_parametervalue = 
  p3023sub3_objflags = 0
  p3023sub4_parametername = PTP.continue
  p3023sub4_objecttype = 7
  p3023sub4_datatype = 6
  p3023sub4_lowlimit = 
  p3023sub4_highlimit = 
  p3023sub4_accesstype = rw
  p3023sub4_pdomapping = 0
  p3023sub4_parametervalue = 
  p3023sub4_objflags = 0
  p3023sub5_parametername = PTP.v_tarPTP
  p3023sub5_objecttype = 7
  p3023sub5_datatype = 6
  p3023sub5_accesstype = rw
  p3023sub5_pdomapping = 0
  p3023sub5_parametervalue = 
  p3023sub5_objflags = 0
  p3024_parametername = vel
  p3024_objecttype = 9
  p3024_subnumber = 0x3
  p3024_parametervalue = 
  p3024_objflags = 0
  p3024sub0_parametername = number of entries
  p3024sub0_objecttype = 7
  p3024sub0_datatype = 5
  p3024sub0_accesstype = ro
  p3024sub0_pdomapping = 0
  p3024sub1_parametername = VEL.velocity
  p3024sub1_objecttype = 7
  p3024sub1_datatype = 3
  p3024sub1_accesstype = rw
  p3024sub1_pdomapping = 0
  p3024sub1_parametervalue = 
  p3024sub1_objflags = 0
  p3024sub2_parametername = VEL.stateVEL
  p3024sub2_objecttype = 7
  p3024sub2_datatype = 6
  p3024sub2_lowlimit = 
  p3024sub2_highlimit = 
  p3024sub2_accesstype = ro
  p3024sub2_pdomapping = 0
  p3028_parametername = homing
  p3028_objecttype = 9
  p3028_subnumber = 0xB
  p3028_parametervalue = 
  p3028_objflags = 0
  p3028sub0_parametername = number of entries
  p3028sub0_objecttype = 7
  p3028sub0_datatype = 5
  p3028sub0_accesstype = ro
  p3028sub0_pdomapping = 0
  p3028sub1_parametername = Homing.startHome
  p3028sub1_objecttype = 7
  p3028sub1_datatype = 6
  p3028sub1_lowlimit = 
  p3028sub1_highlimit = 
  p3028sub1_accesstype = rw
  p3028sub1_pdomapping = 0
  p3028sub1_parametervalue = 
  p3028sub1_objflags = 0
  p3028sub2_parametername = Homing.stateHome
  p3028sub2_objecttype = 7
  p3028sub2_datatype = 6
  p3028sub2_lowlimit = 
  p3028sub2_highlimit = 
  p3028sub2_accesstype = ro
  p3028sub2_pdomapping = 0
  p3028sub3_parametername = Homing.startSetp
  p3028sub3_objecttype = 7
  p3028sub3_datatype = 4
  p3028sub3_lowlimit = 
  p3028sub3_highlimit = 
  p3028sub3_accesstype = rw
  p3028sub3_pdomapping = 0
  p3028sub3_parametervalue = 
  p3028sub3_objflags = 0
  p3028sub4_parametername = Homing.v_Home
  p3028sub4_objecttype = 7
  p3028sub4_datatype = 6
  p3028sub4_accesstype = rw
  p3028sub4_pdomapping = 0
  p3028sub4_parametervalue = 
  p3028sub4_objflags = 0
  p3028sub5_parametername = Homing.v_outHome
  p3028sub5_objecttype = 7
  p3028sub5_datatype = 6
  p3028sub5_accesstype = rw
  p3028sub5_pdomapping = 0
  p3028sub5_parametervalue = 
  p3028sub5_objflags = 0
  p3028sub6_parametername = Homing.p_outHome
  p3028sub6_objecttype = 7
  p3028sub6_datatype = 4
  p3028sub6_lowlimit = 
  p3028sub6_highlimit = 
  p3028sub6_accesstype = rw
  p3028sub6_pdomapping = 0
  p3028sub6_parametervalue = 
  p3028sub6_objflags = 0
  p3028sub7_parametername = Homing.p_disHome
  p3028sub7_objecttype = 7
  p3028sub7_datatype = 4
  p3028sub7_lowlimit = 
  p3028sub7_highlimit = 
  p3028sub7_accesstype = rw
  p3028sub7_pdomapping = 0
  p3028sub7_parametervalue = 
  p3028sub7_objflags = 0
  p3028sub9_parametername = Homing.RefSwMod
  p3028sub9_objecttype = 7
  p3028sub9_datatype = 6
  p3028sub9_lowlimit = 
  p3028sub9_highlimit = 
  p3028sub9_accesstype = rw
  p3028sub9_pdomapping = 0
  p3028sub9_parametervalue = 
  p3028sub9_objflags = 0
  p3028subb_parametername = Homing.RefAppPos
  p3028subb_objecttype = 7
  p3028subb_datatype = 4
  p3028subb_lowlimit = 
  p3028subb_highlimit = 
  p3028subb_accesstype = rw
  p3028subb_pdomapping = 0
  p3028subb_parametervalue = 
  p3028subb_objflags = 0
  p3028subd_parametername = Homing.refError
  p3028subd_objecttype = 7
  p3028subd_datatype = 6
  p3028subd_lowlimit = 
  p3028subd_highlimit = 
  p3028subd_accesstype = ro
  p3028subd_pdomapping = 0
  p3029_parametername = manual
  p3029_objecttype = 9
  p3029_subnumber = 0x7
  p3029_parametervalue = 
  p3029_objflags = 0
  p3029sub0_parametername = number of entries
  p3029sub0_objecttype = 7
  p3029sub0_datatype = 5
  p3029sub0_accesstype = ro
  p3029sub0_pdomapping = 0
  p3029sub1_parametername = Manual.startMan
  p3029sub1_objecttype = 7
  p3029sub1_datatype = 6
  p3029sub1_lowlimit = 
  p3029sub1_highlimit = 
  p3029sub1_accesstype = rw
  p3029sub1_pdomapping = 0
  p3029sub1_parametervalue = 
  p3029sub1_objflags = 0
  p3029sub2_parametername = Manual.stateMan
  p3029sub2_objecttype = 7
  p3029sub2_datatype = 6
  p3029sub2_lowlimit = 
  p3029sub2_highlimit = 
  p3029sub2_accesstype = ro
  p3029sub2_pdomapping = 0
  p3029sub4_parametername = Manual.n_slowMan
  p3029sub4_objecttype = 7
  p3029sub4_datatype = 6
  p3029sub4_accesstype = rw
  p3029sub4_pdomapping = 0
  p3029sub4_parametervalue = 
  p3029sub4_objflags = 0
  p3029sub5_parametername = Manual.n_fastMan
  p3029sub5_objecttype = 7
  p3029sub5_datatype = 6
  p3029sub5_accesstype = rw
  p3029sub5_pdomapping = 0
  p3029sub5_parametervalue = 
  p3029sub5_objflags = 0
  p3029sub7_parametername = Manual.step_Man
  p3029sub7_objecttype = 7
  p3029sub7_datatype = 6
  p3029sub7_lowlimit = 
  p3029sub7_highlimit = 
  p3029sub7_accesstype = rw
  p3029sub7_pdomapping = 0
  p3029sub7_parametervalue = 
  p3029sub7_objflags = 0
  p3029sub8_parametername = Manual.time_Man
  p3029sub8_objecttype = 7
  p3029sub8_datatype = 6
  p3029sub8_lowlimit = 
  p3029sub8_highlimit = 
  p3029sub8_accesstype = rw
  p3029sub8_pdomapping = 0
  p3029sub8_parametervalue = 
  p3029sub8_objflags = 0
  p3320_parametername = prog io0
  p3320_objecttype = 9
  p3320_subnumber = 0x7
  p3320_parametervalue = 
  p3320_objflags = 0
  p3320sub0_parametername = number of entries
  p3320sub0_objecttype = 7
  p3320sub0_datatype = 5
  p3320sub0_accesstype = ro
  p3320sub0_pdomapping = 0
  p3320sub1_parametername = ProgIO0.Index
  p3320sub1_objecttype = 7
  p3320sub1_datatype = 6
  p3320sub1_lowlimit = 
  p3320sub1_highlimit = 
  p3320sub1_accesstype = rw
  p3320sub1_pdomapping = 0
  p3320sub1_parametervalue = 
  p3320sub1_objflags = 0
  p3320sub2_parametername = ProgIO0.Subindex
  p3320sub2_objecttype = 7
  p3320sub2_datatype = 6
  p3320sub2_lowlimit = 
  p3320sub2_highlimit = 
  p3320sub2_accesstype = rw
  p3320sub2_pdomapping = 0
  p3320sub2_parametervalue = 
  p3320sub2_objflags = 0
  p3320sub3_parametername = ProgIO0.BitMask
  p3320sub3_objecttype = 7
  p3320sub3_datatype = 7
  p3320sub3_lowlimit = 
  p3320sub3_highlimit = 
  p3320sub3_accesstype = rw
  p3320sub3_pdomapping = 0
  p3320sub3_parametervalue = 
  p3320sub3_objflags = 0
  p3320sub4_parametername = ProgIO0.Switch
  p3320sub4_objecttype = 7
  p3320sub4_datatype = 6
  p3320sub4_lowlimit = 
  p3320sub4_highlimit = 
  p3320sub4_accesstype = rw
  p3320sub4_pdomapping = 0
  p3320sub4_parametervalue = 
  p3320sub4_objflags = 0
  p3320sub5_parametername = ProgIO0.Value1
  p3320sub5_objecttype = 7
  p3320sub5_datatype = 4
  p3320sub5_lowlimit = 
  p3320sub5_highlimit = 
  p3320sub5_accesstype = rw
  p3320sub5_pdomapping = 0
  p3320sub5_parametervalue = 
  p3320sub5_objflags = 0
  p3320sub6_parametername = ProgIO0.Value2
  p3320sub6_objecttype = 7
  p3320sub6_datatype = 4
  p3320sub6_lowlimit = 
  p3320sub6_highlimit = 
  p3320sub6_accesstype = rw
  p3320sub6_pdomapping = 0
  p3320sub6_parametervalue = 
  p3320sub6_objflags = 0
  p3321_parametername = prog io1
  p3321_objecttype = 9
  p3321_subnumber = 0x7
  p3321_parametervalue = 
  p3321_objflags = 0
  p3321sub0_parametername = number of entries
  p3321sub0_objecttype = 7
  p3321sub0_datatype = 5
  p3321sub0_accesstype = ro
  p3321sub0_pdomapping = 0
  p3321sub1_parametername = ProgIO1.Index
  p3321sub1_objecttype = 7
  p3321sub1_datatype = 6
  p3321sub1_lowlimit = 
  p3321sub1_highlimit = 
  p3321sub1_accesstype = rw
  p3321sub1_pdomapping = 0
  p3321sub1_parametervalue = 
  p3321sub1_objflags = 0
  p3321sub2_parametername = ProgIO1.Subindex
  p3321sub2_objecttype = 7
  p3321sub2_datatype = 6
  p3321sub2_lowlimit = 
  p3321sub2_highlimit = 
  p3321sub2_accesstype = rw
  p3321sub2_pdomapping = 0
  p3321sub2_parametervalue = 
  p3321sub2_objflags = 0
  p3321sub3_parametername = ProgIO1.BitMask
  p3321sub3_objecttype = 7
  p3321sub3_datatype = 7
  p3321sub3_lowlimit = 
  p3321sub3_highlimit = 
  p3321sub3_accesstype = rw
  p3321sub3_pdomapping = 0
  p3321sub3_parametervalue = 
  p3321sub3_objflags = 0
  p3321sub4_parametername = ProgIO1.Switch
  p3321sub4_objecttype = 7
  p3321sub4_datatype = 6
  p3321sub4_lowlimit = 
  p3321sub4_highlimit = 
  p3321sub4_accesstype = rw
  p3321sub4_pdomapping = 0
  p3321sub4_parametervalue = 
  p3321sub4_objflags = 0
  p3321sub5_parametername = ProgIO1.Value1
  p3321sub5_objecttype = 7
  p3321sub5_datatype = 4
  p3321sub5_lowlimit = 
  p3321sub5_highlimit = 
  p3321sub5_accesstype = rw
  p3321sub5_pdomapping = 0
  p3321sub5_parametervalue = 
  p3321sub5_objflags = 0
  p3321sub6_parametername = ProgIO1.Value2
  p3321sub6_objecttype = 7
  p3321sub6_datatype = 4
  p3321sub6_lowlimit = 
  p3321sub6_highlimit = 
  p3321sub6_accesstype = rw
  p3321sub6_pdomapping = 0
  p3321sub6_parametervalue = 
  p3321sub6_objflags = 0
  p3322_parametername = prog io2
  p3322_objecttype = 9
  p3322_subnumber = 0x7
  p3322_parametervalue = 
  p3322_objflags = 0
  p3322sub0_parametername = number of entries
  p3322sub0_objecttype = 7
  p3322sub0_datatype = 5
  p3322sub0_accesstype = ro
  p3322sub0_pdomapping = 0
  p3322sub1_parametername = ProgIO2.Index
  p3322sub1_objecttype = 7
  p3322sub1_datatype = 6
  p3322sub1_lowlimit = 
  p3322sub1_highlimit = 
  p3322sub1_accesstype = rw
  p3322sub1_pdomapping = 0
  p3322sub1_parametervalue = 
  p3322sub1_objflags = 0
  p3322sub2_parametername = ProgIO2.Subindex
  p3322sub2_objecttype = 7
  p3322sub2_datatype = 6
  p3322sub2_lowlimit = 
  p3322sub2_highlimit = 
  p3322sub2_accesstype = rw
  p3322sub2_pdomapping = 0
  p3322sub2_parametervalue = 
  p3322sub2_objflags = 0
  p3322sub3_parametername = ProgIO2.BitMask
  p3322sub3_objecttype = 7
  p3322sub3_datatype = 7
  p3322sub3_lowlimit = 
  p3322sub3_highlimit = 
  p3322sub3_accesstype = rw
  p3322sub3_pdomapping = 0
  p3322sub3_parametervalue = 
  p3322sub3_objflags = 0
  p3322sub4_parametername = ProgIO2.Switch
  p3322sub4_objecttype = 7
  p3322sub4_datatype = 6
  p3322sub4_lowlimit = 
  p3322sub4_highlimit = 
  p3322sub4_accesstype = rw
  p3322sub4_pdomapping = 0
  p3322sub4_parametervalue = 
  p3322sub4_objflags = 0
  p3322sub5_parametername = ProgIO2.Value1
  p3322sub5_objecttype = 7
  p3322sub5_datatype = 4
  p3322sub5_lowlimit = 
  p3322sub5_highlimit = 
  p3322sub5_accesstype = rw
  p3322sub5_pdomapping = 0
  p3322sub5_parametervalue = 
  p3322sub5_objflags = 0
  p3322sub6_parametername = ProgIO2.Value2
  p3322sub6_objecttype = 7
  p3322sub6_datatype = 4
  p3322sub6_lowlimit = 
  p3322sub6_highlimit = 
  p3322sub6_accesstype = rw
  p3322sub6_pdomapping = 0
  p3322sub6_parametervalue = 
  p3322sub6_objflags = 0
  p3323_parametername = prog io3
  p3323_objecttype = 9
  p3323_subnumber = 0x7
  p3323_parametervalue = 
  p3323_objflags = 0
  p3323sub0_parametername = number of entries
  p3323sub0_objecttype = 7
  p3323sub0_datatype = 5
  p3323sub0_accesstype = ro
  p3323sub0_pdomapping = 0
  p3323sub1_parametername = ProgIO3.Index
  p3323sub1_objecttype = 7
  p3323sub1_datatype = 6
  p3323sub1_lowlimit = 
  p3323sub1_highlimit = 
  p3323sub1_accesstype = rw
  p3323sub1_pdomapping = 0
  p3323sub1_parametervalue = 
  p3323sub1_objflags = 0
  p3323sub2_parametername = ProgIO3.Subindex
  p3323sub2_objecttype = 7
  p3323sub2_datatype = 6
  p3323sub2_lowlimit = 
  p3323sub2_highlimit = 
  p3323sub2_accesstype = rw
  p3323sub2_pdomapping = 0
  p3323sub2_parametervalue = 
  p3323sub2_objflags = 0
  p3323sub3_parametername = ProgIO3.BitMask
  p3323sub3_objecttype = 7
  p3323sub3_datatype = 7
  p3323sub3_lowlimit = 
  p3323sub3_highlimit = 
  p3323sub3_accesstype = rw
  p3323sub3_pdomapping = 0
  p3323sub3_parametervalue = 
  p3323sub3_objflags = 0
  p3323sub4_parametername = ProgIO3.Switch
  p3323sub4_objecttype = 7
  p3323sub4_datatype = 6
  p3323sub4_lowlimit = 
  p3323sub4_highlimit = 
  p3323sub4_accesstype = rw
  p3323sub4_pdomapping = 0
  p3323sub4_parametervalue = 
  p3323sub4_objflags = 0
  p3323sub5_parametername = ProgIO3.Value1
  p3323sub5_objecttype = 7
  p3323sub5_datatype = 4
  p3323sub5_lowlimit = 
  p3323sub5_highlimit = 
  p3323sub5_accesstype = rw
  p3323sub5_pdomapping = 0
  p3323sub5_parametervalue = 
  p3323sub5_objflags = 0
  p3323sub6_parametername = ProgIO3.Value2
  p3323sub6_objecttype = 7
  p3323sub6_datatype = 4
  p3323sub6_lowlimit = 
  p3323sub6_highlimit = 
  p3323sub6_accesstype = rw
  p3323sub6_pdomapping = 0
  p3323sub6_parametervalue = 
  p3323sub6_objflags = 0
SI_unit_BK1 : FBC.0x00000114.0x00000003.ex250sca1a_v3.0 v3.0 (OrderNumber=SI unit)  [CAN1 -> ILE1F_BK1.CAN2 (NodeNumber=6)]
  pheartbeat_producertime = 1000
  p2000_parametername = Reserved
  p2000_objecttype = 7
  p2000_datatype = 7
  p2000_accesstype = ro
  p2000_pdomapping = 0
  p2001_parametername = Password
  p2001_objecttype = 7
  p2001_datatype = 6
  p2001_accesstype = wo
  p2001_pdomapping = 0
  p2001_parametervalue = 
  p2001_objflags = 0
  p6000_subnumber = 5
  p6000_parametername = Read Input 8Bit
  p6000_objecttype = 8
  p6000_parametervalue = 
  p6000_objflags = 0
  p6000sub0_parametername = Number of Input 8Bit
  p6000sub0_objecttype = 7
  p6000sub0_datatype = 5
  p6000sub0_accesstype = ro
  p6000sub0_pdomapping = 0
  p6100_subnumber = 3
  p6100_parametername = Read Input 16Bit
  p6100_objecttype = 8
  p6100_parametervalue = 
  p6100_objflags = 0
  p6100sub0_parametername = Number of Input 16Bit
  p6100sub0_objecttype = 7
  p6100sub0_datatype = 5
  p6100sub0_accesstype = ro
  p6100sub0_pdomapping = 0
  p6120_subnumber = 2
  p6120_parametername = Read Input 32Bit
  p6120_objecttype = 8
  p6120_parametervalue = 
  p6120_objflags = 0
  p6120sub0_parametername = Number of Input 32Bit
  p6120sub0_objecttype = 7
  p6120sub0_datatype = 5
  p6120sub0_accesstype = ro
  p6120sub0_pdomapping = 0
  p6200_subnumber = 5
  p6200_parametername = Write Output 8Bit
  p6200_objecttype = 8
  p6200_parametervalue = 
  p6200_objflags = 0
  p6200sub0_parametername = Number of Output 8Bit
  p6200sub0_objecttype = 7
  p6200sub0_datatype = 5
  p6200sub0_accesstype = ro
  p6200sub0_pdomapping = 0
  p6206_subnumber = 5
  p6206_parametername = Error Mode Output 8Bit
  p6206_objecttype = 8
  p6206_parametervalue = 
  p6206_objflags = 0
  p6206sub0_parametername = Number of Output 8Bit
  p6206sub0_objecttype = 7
  p6206sub0_datatype = 5
  p6206sub0_accesstype = ro
  p6206sub0_pdomapping = 0
  p6206sub1_parametername = Error Mode Output 1h to 8h
  p6206sub1_objecttype = 7
  p6206sub1_datatype = 5
  p6206sub1_accesstype = rww
  p6206sub1_pdomapping = 0
  p6206sub1_parametervalue = 0xFF
  p6206sub1_objflags = 0
  p6206sub2_parametername = Error Mode Output 9h to 16h
  p6206sub2_objecttype = 7
  p6206sub2_datatype = 5
  p6206sub2_accesstype = rww
  p6206sub2_pdomapping = 0
  p6206sub2_parametervalue = 0xFF
  p6206sub2_objflags = 0
  p6206sub3_parametername = Error Mode Output 17h to 24h
  p6206sub3_objecttype = 7
  p6206sub3_datatype = 5
  p6206sub3_accesstype = rww
  p6206sub3_pdomapping = 0
  p6206sub3_parametervalue = 0xFF
  p6206sub3_objflags = 0
  p6206sub4_parametername = Error Mode Output 25h to 32h
  p6206sub4_objecttype = 7
  p6206sub4_datatype = 5
  p6206sub4_accesstype = rww
  p6206sub4_pdomapping = 0
  p6206sub4_parametervalue = 0xFF
  p6206sub4_objflags = 0
  p6207_subnumber = 5
  p6207_parametername = Error Value Output 8Bit
  p6207_objecttype = 8
  p6207_parametervalue = 
  p6207_objflags = 0
  p6207sub0_parametername = Number of Output 8Bit
  p6207sub0_objecttype = 7
  p6207sub0_datatype = 5
  p6207sub0_accesstype = ro
  p6207sub0_pdomapping = 0
  p6207sub1_parametername = Error Value Output 1h to 8h
  p6207sub1_objecttype = 7
  p6207sub1_datatype = 5
  p6207sub1_accesstype = rw
  p6207sub1_pdomapping = 0
  p6207sub1_parametervalue = 0x00
  p6207sub1_objflags = 0
  p6207sub2_parametername = Error Value Output 9h to 16h
  p6207sub2_objecttype = 7
  p6207sub2_datatype = 5
  p6207sub2_accesstype = rw
  p6207sub2_pdomapping = 0
  p6207sub2_parametervalue = 0x00
  p6207sub2_objflags = 0
  p6207sub3_parametername = Error Value Output 17h to 24h
  p6207sub3_objecttype = 7
  p6207sub3_datatype = 5
  p6207sub3_accesstype = rw
  p6207sub3_pdomapping = 0
  p6207sub3_parametervalue = 0x00
  p6207sub3_objflags = 0
  p6207sub4_parametername = Error Value Output 25h to 32h
  p6207sub4_objecttype = 7
  p6207sub4_datatype = 5
  p6207sub4_accesstype = rw
  p6207sub4_pdomapping = 0
  p6207sub4_parametervalue = 0x00
  p6207sub4_objflags = 0
  p6300_subnumber = 3
  p6300_parametername = Write Output 16Bit
  p6300_objecttype = 8
  p6300_parametervalue = 
  p6300_objflags = 0
  p6300sub0_parametername = Number of Output 16Bit
  p6300sub0_objecttype = 7
  p6300sub0_datatype = 5
  p6300sub0_accesstype = ro
  p6300sub0_pdomapping = 0
  p6306_subnumber = 3
  p6306_parametername = Error Mode Output 16Bit
  p6306_objecttype = 8
  p6306_parametervalue = 
  p6306_objflags = 0
  p6306sub0_parametername = Number of Output 16Bit
  p6306sub0_objecttype = 7
  p6306sub0_datatype = 5
  p6306sub0_accesstype = ro
  p6306sub0_pdomapping = 0
  p6306sub1_parametername = Error Mode Output 1h to 16h
  p6306sub1_objecttype = 7
  p6306sub1_datatype = 6
  p6306sub1_accesstype = rww
  p6306sub1_pdomapping = 0
  p6306sub1_parametervalue = 0xFFFF
  p6306sub1_objflags = 0
  p6306sub2_parametername = Error Mode Output 17h to 32h
  p6306sub2_objecttype = 7
  p6306sub2_datatype = 6
  p6306sub2_accesstype = rww
  p6306sub2_pdomapping = 0
  p6306sub2_parametervalue = 0xFFFF
  p6306sub2_objflags = 0
  p6307_subnumber = 3
  p6307_parametername = Error Value Output 16Bit
  p6307_objecttype = 8
  p6307_parametervalue = 
  p6307_objflags = 0
  p6307sub0_parametername = Number of Output 16Bit
  p6307sub0_objecttype = 7
  p6307sub0_datatype = 5
  p6307sub0_accesstype = ro
  p6307sub0_pdomapping = 0
  p6307sub1_parametername = Error Value Output 1h to 16h
  p6307sub1_objecttype = 7
  p6307sub1_datatype = 6
  p6307sub1_accesstype = rw
  p6307sub1_pdomapping = 0
  p6307sub1_parametervalue = 0x0000
  p6307sub1_objflags = 0
  p6307sub2_parametername = Error Value Output 17h to 32h
  p6307sub2_objecttype = 7
  p6307sub2_datatype = 6
  p6307sub2_accesstype = rw
  p6307sub2_pdomapping = 0
  p6307sub2_parametervalue = 0x0000
  p6307sub2_objflags = 0
  p6320_subnumber = 2
  p6320_parametername = Write Output 32Bit
  p6320_objecttype = 8
  p6320_parametervalue = 
  p6320_objflags = 0
  p6320sub0_parametername = Number of Output 32Bit
  p6320sub0_objecttype = 7
  p6320sub0_datatype = 5
  p6320sub0_accesstype = ro
  p6320sub0_pdomapping = 0
  p6326_subnumber = 2
  p6326_parametername = Error Mode Output 32Bit
  p6326_objecttype = 8
  p6326_parametervalue = 
  p6326_objflags = 0
  p6326sub0_parametername = Number of Output 32Bit
  p6326sub0_objecttype = 7
  p6326sub0_datatype = 5
  p6326sub0_accesstype = ro
  p6326sub0_pdomapping = 0
  p6326sub1_parametername = Error Mode Output 1h to 32h
  p6326sub1_objecttype = 7
  p6326sub1_datatype = 7
  p6326sub1_accesstype = rww
  p6326sub1_pdomapping = 0
  p6326sub1_parametervalue = 0xFFFFFFFF
  p6326sub1_objflags = 0
  p6327_subnumber = 2
  p6327_parametername = Error Value Output 32Bit
  p6327_objecttype = 8
  p6327_parametervalue = 
  p6327_objflags = 0
  p6327sub0_parametername = Number of Output 32Bit
  p6327sub0_objecttype = 7
  p6327sub0_datatype = 5
  p6327sub0_accesstype = ro
  p6327sub0_pdomapping = 0
  p6327sub1_parametername = Error Value Output 1h to 32h
  p6327sub1_objecttype = 7
  p6327sub1_datatype = 7
  p6327sub1_accesstype = rw
  p6327sub1_pdomapping = 0
  p6327sub1_parametervalue = 0x00000000
  p6327sub1_objflags = 0
SI_unit_BK2 : FBC.0x00000114.0x00000003.ex250sca1a_v3.0 v3.0 (OrderNumber=SI unit)  [CAN1 -> ILE1F_BK2.CAN2 (NodeNumber=8)]
  pheartbeat_producertime = 1000
  p2000_parametername = Reserved
  p2000_objecttype = 7
  p2000_datatype = 7
  p2000_accesstype = ro
  p2000_pdomapping = 0
  p2001_parametername = Password
  p2001_objecttype = 7
  p2001_datatype = 6
  p2001_accesstype = wo
  p2001_pdomapping = 0
  p2001_parametervalue = 
  p2001_objflags = 0
  p6000_subnumber = 5
  p6000_parametername = Read Input 8Bit
  p6000_objecttype = 8
  p6000_parametervalue = 
  p6000_objflags = 0
  p6000sub0_parametername = Number of Input 8Bit
  p6000sub0_objecttype = 7
  p6000sub0_datatype = 5
  p6000sub0_accesstype = ro
  p6000sub0_pdomapping = 0
  p6100_subnumber = 3
  p6100_parametername = Read Input 16Bit
  p6100_objecttype = 8
  p6100_parametervalue = 
  p6100_objflags = 0
  p6100sub0_parametername = Number of Input 16Bit
  p6100sub0_objecttype = 7
  p6100sub0_datatype = 5
  p6100sub0_accesstype = ro
  p6100sub0_pdomapping = 0
  p6120_subnumber = 2
  p6120_parametername = Read Input 32Bit
  p6120_objecttype = 8
  p6120_parametervalue = 
  p6120_objflags = 0
  p6120sub0_parametername = Number of Input 32Bit
  p6120sub0_objecttype = 7
  p6120sub0_datatype = 5
  p6120sub0_accesstype = ro
  p6120sub0_pdomapping = 0
  p6200_subnumber = 5
  p6200_parametername = Write Output 8Bit
  p6200_objecttype = 8
  p6200_parametervalue = 
  p6200_objflags = 0
  p6200sub0_parametername = Number of Output 8Bit
  p6200sub0_objecttype = 7
  p6200sub0_datatype = 5
  p6200sub0_accesstype = ro
  p6200sub0_pdomapping = 0
  p6206_subnumber = 5
  p6206_parametername = Error Mode Output 8Bit
  p6206_objecttype = 8
  p6206_parametervalue = 
  p6206_objflags = 0
  p6206sub0_parametername = Number of Output 8Bit
  p6206sub0_objecttype = 7
  p6206sub0_datatype = 5
  p6206sub0_accesstype = ro
  p6206sub0_pdomapping = 0
  p6206sub1_parametername = Error Mode Output 1h to 8h
  p6206sub1_objecttype = 7
  p6206sub1_datatype = 5
  p6206sub1_accesstype = rww
  p6206sub1_pdomapping = 0
  p6206sub1_parametervalue = 0xFF
  p6206sub1_objflags = 0
  p6206sub2_parametername = Error Mode Output 9h to 16h
  p6206sub2_objecttype = 7
  p6206sub2_datatype = 5
  p6206sub2_accesstype = rww
  p6206sub2_pdomapping = 0
  p6206sub2_parametervalue = 0xFF
  p6206sub2_objflags = 0
  p6206sub3_parametername = Error Mode Output 17h to 24h
  p6206sub3_objecttype = 7
  p6206sub3_datatype = 5
  p6206sub3_accesstype = rww
  p6206sub3_pdomapping = 0
  p6206sub3_parametervalue = 0xFF
  p6206sub3_objflags = 0
  p6206sub4_parametername = Error Mode Output 25h to 32h
  p6206sub4_objecttype = 7
  p6206sub4_datatype = 5
  p6206sub4_accesstype = rww
  p6206sub4_pdomapping = 0
  p6206sub4_parametervalue = 0xFF
  p6206sub4_objflags = 0
  p6207_subnumber = 5
  p6207_parametername = Error Value Output 8Bit
  p6207_objecttype = 8
  p6207_parametervalue = 
  p6207_objflags = 0
  p6207sub0_parametername = Number of Output 8Bit
  p6207sub0_objecttype = 7
  p6207sub0_datatype = 5
  p6207sub0_accesstype = ro
  p6207sub0_pdomapping = 0
  p6207sub1_parametername = Error Value Output 1h to 8h
  p6207sub1_objecttype = 7
  p6207sub1_datatype = 5
  p6207sub1_accesstype = rw
  p6207sub1_pdomapping = 0
  p6207sub1_parametervalue = 0x00
  p6207sub1_objflags = 0
  p6207sub2_parametername = Error Value Output 9h to 16h
  p6207sub2_objecttype = 7
  p6207sub2_datatype = 5
  p6207sub2_accesstype = rw
  p6207sub2_pdomapping = 0
  p6207sub2_parametervalue = 0x00
  p6207sub2_objflags = 0
  p6207sub3_parametername = Error Value Output 17h to 24h
  p6207sub3_objecttype = 7
  p6207sub3_datatype = 5
  p6207sub3_accesstype = rw
  p6207sub3_pdomapping = 0
  p6207sub3_parametervalue = 0x00
  p6207sub3_objflags = 0
  p6207sub4_parametername = Error Value Output 25h to 32h
  p6207sub4_objecttype = 7
  p6207sub4_datatype = 5
  p6207sub4_accesstype = rw
  p6207sub4_pdomapping = 0
  p6207sub4_parametervalue = 0x00
  p6207sub4_objflags = 0
  p6300_subnumber = 3
  p6300_parametername = Write Output 16Bit
  p6300_objecttype = 8
  p6300_parametervalue = 
  p6300_objflags = 0
  p6300sub0_parametername = Number of Output 16Bit
  p6300sub0_objecttype = 7
  p6300sub0_datatype = 5
  p6300sub0_accesstype = ro
  p6300sub0_pdomapping = 0
  p6306_subnumber = 3
  p6306_parametername = Error Mode Output 16Bit
  p6306_objecttype = 8
  p6306_parametervalue = 
  p6306_objflags = 0
  p6306sub0_parametername = Number of Output 16Bit
  p6306sub0_objecttype = 7
  p6306sub0_datatype = 5
  p6306sub0_accesstype = ro
  p6306sub0_pdomapping = 0
  p6306sub1_parametername = Error Mode Output 1h to 16h
  p6306sub1_objecttype = 7
  p6306sub1_datatype = 6
  p6306sub1_accesstype = rww
  p6306sub1_pdomapping = 0
  p6306sub1_parametervalue = 0xFFFF
  p6306sub1_objflags = 0
  p6306sub2_parametername = Error Mode Output 17h to 32h
  p6306sub2_objecttype = 7
  p6306sub2_datatype = 6
  p6306sub2_accesstype = rww
  p6306sub2_pdomapping = 0
  p6306sub2_parametervalue = 0xFFFF
  p6306sub2_objflags = 0
  p6307_subnumber = 3
  p6307_parametername = Error Value Output 16Bit
  p6307_objecttype = 8
  p6307_parametervalue = 
  p6307_objflags = 0
  p6307sub0_parametername = Number of Output 16Bit
  p6307sub0_objecttype = 7
  p6307sub0_datatype = 5
  p6307sub0_accesstype = ro
  p6307sub0_pdomapping = 0
  p6307sub1_parametername = Error Value Output 1h to 16h
  p6307sub1_objecttype = 7
  p6307sub1_datatype = 6
  p6307sub1_accesstype = rw
  p6307sub1_pdomapping = 0
  p6307sub1_parametervalue = 0x0000
  p6307sub1_objflags = 0
  p6307sub2_parametername = Error Value Output 17h to 32h
  p6307sub2_objecttype = 7
  p6307sub2_datatype = 6
  p6307sub2_accesstype = rw
  p6307sub2_pdomapping = 0
  p6307sub2_parametervalue = 0x0000
  p6307sub2_objflags = 0
  p6320_subnumber = 2
  p6320_parametername = Write Output 32Bit
  p6320_objecttype = 8
  p6320_parametervalue = 
  p6320_objflags = 0
  p6320sub0_parametername = Number of Output 32Bit
  p6320sub0_objecttype = 7
  p6320sub0_datatype = 5
  p6320sub0_accesstype = ro
  p6320sub0_pdomapping = 0
  p6326_subnumber = 2
  p6326_parametername = Error Mode Output 32Bit
  p6326_objecttype = 8
  p6326_parametervalue = 
  p6326_objflags = 0
  p6326sub0_parametername = Number of Output 32Bit
  p6326sub0_objecttype = 7
  p6326sub0_datatype = 5
  p6326sub0_accesstype = ro
  p6326sub0_pdomapping = 0
  p6326sub1_parametername = Error Mode Output 1h to 32h
  p6326sub1_objecttype = 7
  p6326sub1_datatype = 7
  p6326sub1_accesstype = rww
  p6326sub1_pdomapping = 0
  p6326sub1_parametervalue = 0xFFFFFFFF
  p6326sub1_objflags = 0
  p6327_subnumber = 2
  p6327_parametername = Error Value Output 32Bit
  p6327_objecttype = 8
  p6327_parametervalue = 
  p6327_objflags = 0
  p6327sub0_parametername = Number of Output 32Bit
  p6327sub0_objecttype = 7
  p6327sub0_datatype = 5
  p6327sub0_accesstype = ro
  p6327sub0_pdomapping = 0
  p6327sub1_parametername = Error Value Output 1h to 32h
  p6327sub1_objecttype = 7
  p6327sub1_datatype = 7
  p6327sub1_accesstype = rw
  p6327sub1_pdomapping = 0
  p6327sub1_parametervalue = 0x00000000
  p6327sub1_objflags = 0
X20AI2636_005 : X20AI2636 v1.2.0.0  [SS1 -> X20TB12j.SS; SL -> X20BM11v.SL1]
  Supervision = off
  ChannelType0x = 0 to 20mA
  SampleTime = 65536000
  Channel02enable = off
  PhysValueDisplay = sampled
  PhysSampleCount = off
  PhySamCh01_0 = on
  PhySamCh01_1 = on
  PhySamCh01_2 = on
  PhySamCh01_3 = on
  PhySamCh01_4 = on
  PhySamCh01_5 = on
  PhySamCh01_6 = on
  PhySamCh01_7 = on
  PhySamCh01_8 = on
  PhySamCh01_9 = on
  PhySamCh01_10 = on
  PhySamCh01_11 = on
  PhySamCh01_12 = on
X20AI8321_109 : X20AI8321 v1.5.0.0  [SS1 -> X20TB1F14.SS; SL -> X20BM11r.SL1]
  Supervision = off
  LowerLimit = -8000  // Specifies the lower measurement limit, this limit changed from -32676 to -8000 because, It is reading -8190 when sensor is disconnected
  ChannelType01 = 4 to 20mA  // Current 0 to 20 mA / current 4 to 20 mA ; P4 is working with current 4 to 20 mA
  ChannelType02 = 4 to 20mA  // Current 0 to 20 mA / current 4 to 20 mA ; P4 is working with current 4 to 20 mA
  ChannelType03 = 4 to 20mA  // Current 0 to 20 mA / current 4 to 20 mA ; P4 is working with current 4 to 20 mA
  ChannelType04 = 4 to 20mA  // Current 0 to 20 mA / current 4 to 20 mA ; P4 is working with current 4 to 20 mA
  ChannelType05 = 4 to 20mA  // Current 0 to 20 mA / current 4 to 20 mA ; P4 is working with current 4 to 20 mA
  ChannelType06 = 4 to 20mA  // Current 0 to 20 mA / current 4 to 20 mA ; P4 is working with current 4 to 20 mA
  ChannelType07 = 4 to 20mA  // Current 0 to 20 mA / current 4 to 20 mA ; P4 is working with current 4 to 20 mA
  ChannelType08 = 4 to 20mA  // Current 0 to 20 mA / current 4 to 20 mA ; P4 is working with current 4 to 20 mA
X20AI8321_110 : X20AI8321 v1.5.0.0  [SS1 -> X20TB1F15.SS; SL -> X20BM11s.SL1]
  Supervision = off
  LowerLimit = -8000  // Specifies the lower measurement limit, this limit changed from -32676 to -8000 because, It is reading -8190 when sensor is disconnected
  ChannelType01 = 4 to 20mA  // Current 0 to 20 mA / current 4 to 20 mA ; P4 is working with current 4 to 20 mA
  ChannelType02 = 4 to 20mA  // Current 0 to 20 mA / current 4 to 20 mA ; P4 is working with current 4 to 20 mA
  ChannelType03 = 4 to 20mA  // Current 0 to 20 mA / current 4 to 20 mA ; P4 is working with current 4 to 20 mA
  ChannelType04 = 4 to 20mA  // Current 0 to 20 mA / current 4 to 20 mA ; P4 is working with current 4 to 20 mA
  ChannelType05 = 4 to 20mA  // Current 0 to 20 mA / current 4 to 20 mA ; P4 is working with current 4 to 20 mA
  ChannelType06 = 4 to 20mA  // Current 0 to 20 mA / current 4 to 20 mA ; P4 is working with current 4 to 20 mA
  ChannelType07 = 4 to 20mA  // Current 0 to 20 mA / current 4 to 20 mA ; P4 is working with current 4 to 20 mA
  ChannelType08 = 4 to 20mA  // Current 0 to 20 mA / current 4 to 20 mA ; P4 is working with current 4 to 20 mA
X20AI8321_209 : X20AI8321 v1.5.0.0  [SS1 -> X20TB1F21.SS; SL -> X20BM11ae.SL1]
  Supervision = off
  LowerLimit = -8000  // Specifies the lower measurement limit, this limit changed from -32676 to -8000 because, It is reading -8190 when sensor is disconnected
  ChannelType01 = 4 to 20mA  // Current 0 to 20 mA / current 4 to 20 mA ; P4 is working with current 4 to 20 mA
  ChannelType02 = 4 to 20mA  // Current 0 to 20 mA / current 4 to 20 mA ; P4 is working with current 4 to 20 mA
  ChannelType03 = 4 to 20mA  // Current 0 to 20 mA / current 4 to 20 mA ; P4 is working with current 4 to 20 mA
  ChannelType04 = 4 to 20mA  // Current 0 to 20 mA / current 4 to 20 mA ; P4 is working with current 4 to 20 mA
  ChannelType05 = 4 to 20mA  // Current 0 to 20 mA / current 4 to 20 mA ; P4 is working with current 4 to 20 mA
  ChannelType06 = 4 to 20mA  // Current 0 to 20 mA / current 4 to 20 mA ; P4 is working with current 4 to 20 mA
  ChannelType07 = 4 to 20mA  // Current 0 to 20 mA / current 4 to 20 mA ; P4 is working with current 4 to 20 mA
  ChannelType08 = 4 to 20mA  // Current 0 to 20 mA / current 4 to 20 mA ; P4 is working with current 4 to 20 mA
X20AI8321_210 : X20AI8321 v1.5.0.0  [SS1 -> X20TB1F22.SS; SL -> X20BM11af.SL1]
  Supervision = off
  LowerLimit = -8000  // Specifies the lower measurement limit, this limit changed from -32676 to -8000 because, It is reading -8190 when sensor is disconnected
  ChannelType01 = 4 to 20mA  // Current 0 to 20 mA / current 4 to 20 mA ; P4 is working with current 4 to 20 mA
  ChannelType02 = 4 to 20mA  // Current 0 to 20 mA / current 4 to 20 mA ; P4 is working with current 4 to 20 mA
  ChannelType03 = 4 to 20mA  // Current 0 to 20 mA / current 4 to 20 mA ; P4 is working with current 4 to 20 mA
  ChannelType04 = 4 to 20mA  // Current 0 to 20 mA / current 4 to 20 mA ; P4 is working with current 4 to 20 mA
  ChannelType05 = 4 to 20mA  // Current 0 to 20 mA / current 4 to 20 mA ; P4 is working with current 4 to 20 mA
  ChannelType06 = 4 to 20mA  // Current 0 to 20 mA / current 4 to 20 mA ; P4 is working with current 4 to 20 mA
  ChannelType07 = 4 to 20mA  // Current 0 to 20 mA / current 4 to 20 mA ; P4 is working with current 4 to 20 mA
  ChannelType08 = 4 to 20mA  // Current 0 to 20 mA / current 4 to 20 mA ; P4 is working with current 4 to 20 mA
X20AO4622_111 : X20AO4622 v1.3.0.0  [SS1 -> X20TB12b.SS; SL -> X20BM11l.SL1]
  Supervision = off
X20AO4622_112 : X20AO4622 v1.3.0.0  [SS1 -> X20TB12c.SS; SL -> X20BM11m.SL1]
  Supervision = off
X20AO4622_113 : X20AO4622 v1.3.0.0  [SS1 -> X20TB12d.SS; SL -> X20BM11n.SL1]
  Supervision = off
X20AO4622_211 : X20AO4622 v1.3.0.0  [SS1 -> X20TB12o.SS; SL -> X20BM11ag.SL1]
  Supervision = off
X20AO4622_212 : X20AO4622 v1.3.0.0  [SS1 -> X20TB12p.SS; SL -> X20BM11ah.SL1]
  Supervision = off
X20AO4622_213 : X20AO4622 v1.3.0.0  [SS1 -> X20TB12q.SS; SL -> X20BM11ai.SL1]
  Supervision = off
X20AT4222_114 : X20AT4222 v1.4.0.0  [SS1 -> X20TB12e.SS; SL -> X20BM11o.SL1]
  Supervision = off
X20AT4222_115 : X20AT4222 v1.4.0.0  [SS1 -> X20TB12f.SS; SL -> X20BM11p.SL1]
  Supervision = off
X20AT4222_116 : X20AT4222 v1.4.0.0  [SS1 -> X20TB12i.SS; SL -> X20BM11u.SL1]
  Supervision = off
X20AT4222_214 : X20AT4222 v1.4.0.0  [SS1 -> X20TB12r.SS; SL -> X20BM11aj.SL1]
  Supervision = off
X20AT4222_215 : X20AT4222 v1.4.0.0  [SS1 -> X20TB12s.SS; SL -> X20BM11ak.SL1]
  Supervision = off
X20AT4222_216 : X20AT4222 v1.4.0.0  [SS1 -> X20TB12t.SS; SL -> X20BM11al.SL1]
  Supervision = off
X20BM01 : X20BM01 v2.2.0.0
X20BM01a : X20BM01 v2.2.0.0
X20BM11 : X20BM11 v1.1.0.0  [X2X1 -> X20CP1382.IF6]
X20BM11a : X20BM11 v1.1.0.0  [X2X1 -> X20BM11.X2X2]
X20BM11aa : X20BM11 v1.1.0.0 (Disabled=true)  [X2X1 -> X20BM11z.X2X2]
X20BM11ab : X20BM11 v1.1.0.0  [X2X1 -> X20BM11aa.X2X2]
X20BM11ac : X20BM11 v1.1.0.0  [X2X1 -> X20BM11ab.X2X2]
X20BM11ad : X20BM11 v1.1.0.0  [X2X1 -> X20BM11ac.X2X2]
X20BM11ae : X20BM11 v1.1.0.0  [X2X1 -> X20BM11ad.X2X2]
X20BM11af : X20BM11 v1.1.0.0  [X2X1 -> X20BM11ae.X2X2]
X20BM11ag : X20BM11 v1.1.0.0  [X2X1 -> X20BM11af.X2X2]
X20BM11ah : X20BM11 v1.1.0.0  [X2X1 -> X20BM11ag.X2X2]
X20BM11ai : X20BM11 v1.1.0.0  [X2X1 -> X20BM11ah.X2X2]
X20BM11aj : X20BM11 v1.1.0.0  [X2X1 -> X20BM11ai.X2X2]
X20BM11ak : X20BM11 v1.1.0.0  [X2X1 -> X20BM11aj.X2X2]
X20BM11al : X20BM11 v1.1.0.0  [X2X1 -> X20BM11ak.X2X2]
X20BM11b : X20BM11 v1.1.0.0  [X2X1 -> X20BM11a.X2X2]
X20BM11c : X20BM11 v1.1.0.0  [X2X1 -> X20BM11b.X2X2]
X20BM11e : X20BM11 v1.1.0.0  [X2X1 -> X20BM01.X2X2]
X20BM11f : X20BM11 v1.1.0.0  [X2X1 -> X20BM11e.X2X2]
X20BM11g : X20BM11 v1.1.0.0  [X2X1 -> X20BM11f.X2X2]
X20BM11h : X20BM11 v1.1.0.0 (Disabled=true)  [X2X1 -> X20BM11g.X2X2]
X20BM11i : X20BM11 v1.1.0.0  [X2X1 -> X20BM11k.X2X2]
X20BM11j : X20BM11 v1.1.0.0  [X2X1 -> X20BM11w.X2X2]
X20BM11k : X20BM11 v1.1.0.0  [X2X1 -> X20BM11j.X2X2]
X20BM11l : X20BM11 v1.1.0.0  [X2X1 -> X20BM11s.X2X2]
X20BM11m : X20BM11 v1.1.0.0  [X2X1 -> X20BM11l.X2X2]
X20BM11n : X20BM11 v1.1.0.0  [X2X1 -> X20BM11m.X2X2]
X20BM11o : X20BM11 v1.1.0.0  [X2X1 -> X20BM11n.X2X2]
X20BM11p : X20BM11 v1.1.0.0  [X2X1 -> X20BM11o.X2X2]
X20BM11q : X20BM11 v1.1.0.0  [X2X1 -> X20BM01a.X2X2]
X20BM11r : X20BM11 v1.1.0.0  [X2X1 -> X20BM11i.X2X2]
X20BM11s : X20BM11 v1.1.0.0  [X2X1 -> X20BM11r.X2X2]
X20BM11u : X20BM11 v1.1.0.0  [X2X1 -> X20BM11p.X2X2]
X20BM11v : X20BM11 v1.1.0.0  [X2X1 -> X20BM11c.X2X2]
X20BM11w : X20BM11 v1.1.0.0 (Disabled=true)  [X2X1 -> X20BM11h.X2X2]
X20BM11x : X20BM11 v1.1.0.0  [X2X1 -> X20BM11q.X2X2]
X20BM11y : X20BM11 v1.1.0.0  [X2X1 -> X20BM11x.X2X2]
X20BM11z : X20BM11 v1.1.0.0 (Disabled=true)  [X2X1 -> X20BM11y.X2X2]
X20BM13 : X20BM13 v1.1.0.0  [X2X1 -> X20BM11u.X2X2]
X20BM13a : X20BM13 v1.1.0.0  [X2X1 -> X20BM11al.X2X2]
X20BM15 : X20BM15 v1.1.0.0  [X2X1 -> X20BM31a.X2X2 (NodeNumber=30)]
X20BM15a : X20BM15 v1.1.0.0  [X2X1 -> X20BM15.X2X2 (NodeNumber=99)]
X20BM15b : X20BM15 v1.1.0.0  [X2X1 -> X20BM33b.X2X2 (NodeNumber=199)]
X20BM31 : X20BM31 v1.1.0.0  [X2X1 -> X20BM33a.X2X2]
X20BM31a : X20BM31 v1.1.0.0  [X2X1 -> X20BM31.X2X2]
X20BM33a : X20BM33 v1.1.0.0  [X2X1 -> X20BM11v.X2X2]
X20BM33b : X20BM33 v1.1.0.0  [X2X1 -> X20BM13.X2X2]
X20BM33c : X20BM33 v1.1.0.0  [X2X1 -> X20BM13a.X2X2]
X20BR9300_100 : X20BR9300 v1.3.0.0  [SS1 -> X20TB12a.SS; SL -> X20BM01.SL1; X2X1 -> X20BT9100_099.X2X1 [Cable Type=X2XCable, Length=10, Version=1.0.0.3]]
  Supervision = off
  StatusInfo = off
X20BR9300_200 : X20BR9300 v1.3.0.0  [SS1 -> X20TB12h.SS; SL -> X20BM01a.SL1; X2X1 -> X20BT9100_199.X2X1 [Cable Type=X2XCable, Length=10, Version=1.0.0.3]]
  Supervision = off
X20BT9100_099 : X20BT9100 v1.3.0.0  [SS1 -> X20TB12.SS; SL -> X20BM15a.SL1]
  Supervision = off
  StatusInfo = off
X20BT9100_199 : X20BT9100 v1.3.0.0  [SS1 -> X20TB12g.SS; SL -> X20BM15b.SL1]
  Supervision = off
X20CP1382 : X20CP1382 v1.14.0.0  [X1 -> X1.SL; X2 -> X2.SL; X3 -> X3.SL]
  Module X1 (Type=X1, Virtual=true, Version=1.14.0.0)
    Connection (Connector=SS1, TargetModule=X20TB1F, TargetConnector=SS)
    Connection (Connector=SL, TargetModule=X20CP1382, TargetConnector=X1)
  Module X2 (Type=X2, Virtual=true, Version=1.14.0.0)
    Connection (Connector=SS1, TargetModule=X20TB1F1, TargetConnector=SS)
    Connection (Connector=SL, TargetModule=X20CP1382, TargetConnector=X2)
  Module X3 (Type=X3, Virtual=true, Version=1.14.0.0)
    Connection (Connector=SS1, TargetModule=X20TB1F2, TargetConnector=SS)
    Connection (Connector=SL, TargetModule=X20CP1382, TargetConnector=X3)
    X3Channel05Config = input
    X3Channel06Config = input
    X3Channel07Config = input
  Connector IF2:
    ActivateDevice = 1
    Mode = Manual
    InternetAddress = 192.168.127.10
    SubnetMask = 255.255.255.0
    InaNodeNumber = 0
    Vnc1
    VncVcObjectName1 = Panel1
    VncKeyMappingFile1 = VC\PS2-Keyboard2.dis
    VncPortNumber1 = 5903
    VncMaxConnections1 = 2
    VncRefreshRate1 = 200
    VncTitle1 = EFI P4 Safety Configuration
  Connector IF3:
    MtuSize = 1000
    DNAConfiguration = manual
    CycleTime = 2000
  Connector IF7:
    Baudrate = 250000
    ActivateCANIO = 0
    ActivateCanOpen = 1
    pnmtstartup_maximumbootuptime = 15
    pnmtstartup_pnptimer = 1
    procPriority = 197
    pheartbeat_producertime = 0
    pheartbeat_securityfactor = 0
    pactivatesync = 1
    pcycleperiod = 10000
    pwindowlength = 10000
    p1006_parametervalue = 0
    p1007_parametervalue = 0
    p100c_parametervalue = 1000
    p100d_parametervalue = 3
  ConfigurationID = 2BK12Bar
  UserPartitionSize = 400
  PermanentPvSize = 25000
  RemanentGlobalPvSize = 5000
  VolatileGlobalPvSize = 500000
  UserLoggerSize = 4096000
  EnableUsbRemoteInstall = 1
  EnableCfRemoteInstall = 1
  TimerDeviceType = EPLX2X
  TimerDevice = X20CP1382.IF3
  IdleTaskClass = 3
  TaskClassIdleTime = 8000
  CyclicTaskClassCount = 7
  Cyclic1Duration = 4000  // In this Cyclic task is located Stepper by X2X commns
  Cyclic1Tolerance = 0
  Cyclic1Stack = 16000
  Cyclic1Output = 1
  Cyclic2Duration = 12000
  Cyclic2Tolerance = 0
  Cyclic3Duration = 16000
  Cyclic3Tolerance = 16000
  Cyclic4Duration = 32000
  Cyclic4Tolerance = 32000
  Cyclic5Duration = 80000
  Cyclic5Tolerance = 80000
  Cyclic6Duration = 88000
  Cyclic6Tolerance = 88000
  Cyclic7Duration = 44000
  Cyclic7Tolerance = 88000
  Cyclic8Duration = 30000000
  TimeZone = 150
  ActivateDaylightSavingTime = 1
  FtpUser1
  FtpUsername1 = EFI  // EFI
  FtpUserPassword1 = slxl0rSrlHol5+f9HDoVQew+NWN2FALixC0tIwzGES4=  // Castellon
  FtpUserSalt1 = yh+eVJGC
  FTPAccessRight1 = 0
  ActivateOpcUa = 1
  OpcUaInformationModels_PV_Version = 1
X20DC4395_104 : X20DC4395 v1.3.0.0 (Disabled=true)  [SS1 -> X20TB12k.SS; SL -> X20BM11h.SL1]
  Supervision = off
  ConfigChannel0104 = Standard
  ConfigChannel0102 = Standard
  Channel01Config = Event
  Channel02Config = Event
  ConfigChannel0304 = Standard
  Channel03Config = Event
  Channel04Config = Event
  ConfigChannel0508 = Standard
  ConfigChannel0506 = Standard
  Channel05Config = Event
  Channel06Config = Event
  ConfigChannel0708 = Standard
  Channel07Config = Event
  Channel08Config = Event
X20DC4395_105 : X20DC4395 v1.3.0.0 (Disabled=true)  [SS1 -> X20TB12l.SS; SL -> X20BM11w.SL1]
  Supervision = off
  ConfigChannel0104 = Standard
  ConfigChannel0102 = Standard
  Channel01Config = Event
  Channel02Config = Event
  ConfigChannel0304 = Standard
  Channel03Config = Event
  Channel04Config = Event
  ConfigChannel0508 = Standard
  ConfigChannel0506 = Standard
  Channel05Config = Event
  Channel06Config = Event
  ConfigChannel0708 = Standard
  Channel07Config = Event
  Channel08Config = Event
X20DC4395_204 : X20DC4395 v1.3.0.0 (Disabled=true)  [SS1 -> X20TB12m.SS; SL -> X20BM11z.SL1]
  Supervision = off
  ConfigChannel0104 = Standard
  ConfigChannel0102 = Standard
  Channel01Config = Event
  Channel02Config = Event
  ConfigChannel0304 = Standard
  Channel03Config = Event
  Channel04Config = Event
  ConfigChannel0508 = Standard
  ConfigChannel0506 = Standard
  Channel05Config = Event
  Channel06Config = Event
  ConfigChannel0708 = Standard
  Channel07Config = Event
  Channel08Config = Event
X20DC4395_205 : X20DC4395 v1.3.0.0 (Disabled=true)  [SS1 -> X20TB12n.SS; SL -> X20BM11aa.SL1]
  Supervision = off
  ConfigChannel0104 = Standard
  ConfigChannel0102 = Standard
  Channel01Config = Event
  Channel02Config = Event
  ConfigChannel0304 = Standard
  Channel03Config = Event
  Channel04Config = Event
  ConfigChannel0508 = Standard
  ConfigChannel0506 = Standard
  Channel05Config = Event
  Channel06Config = Event
  ConfigChannel0708 = Standard
  Channel07Config = Event
  Channel08Config = Event
X20DIF371_002 : X20DIF371 v1.3.0.0  [SS1 -> X20TB1F4.SS; SL -> X20BM11a.SL1]
  Supervision = off
X20DIF371_003 : X20DIF371 v1.3.0.0  [SS1 -> X20TB1F5.SS; SL -> X20BM11b.SL1]
  Supervision = off
X20DIF371_030 : X20DIF371 v1.3.0.0  [SS1 -> X20TB1F23.SS; SL -> X20BM15.SL1]
  Supervision = off
X20DIF371_101 : X20DIF371 v1.3.0.0  [SS1 -> X20TB1F7.SS; SL -> X20BM11e.SL1]
  Supervision = off
X20DIF371_102 : X20DIF371 v1.3.0.0  [SS1 -> X20TB1F8.SS; SL -> X20BM11f.SL1]
  Supervision = off
X20DIF371_103 : X20DIF371 v1.3.0.0  [SS1 -> X20TB1F9.SS; SL -> X20BM11g.SL1]
  Supervision = off
X20DIF371_201 : X20DIF371 v1.3.0.0  [SS1 -> X20TB1F11.SS; SL -> X20BM11q.SL1]
  Supervision = off
X20DIF371_202 : X20DIF371 v1.3.0.0  [SS1 -> X20TB1F16.SS; SL -> X20BM11x.SL1]
  Supervision = off
X20DIF371_203 : X20DIF371 v1.3.0.0  [SS1 -> X20TB1F17.SS; SL -> X20BM11y.SL1]
  Supervision = off
X20DOF322_001 : X20DOF322 v1.5.0.0  [SS1 -> X20TB1F3.SS; SL -> X20BM11.SL1]
  Supervision = off
X20DOF322_004 : X20DOF322 v1.5.0.0  [SS1 -> X20TB1F6.SS; SL -> X20BM11c.SL1]
  Supervision = off
X20DOF322_106 : X20DOF322 v1.5.0.0  [SS1 -> X20TB1F12.SS; SL -> X20BM11j.SL1]
  Supervision = off
X20DOF322_107 : X20DOF322 v1.5.0.0  [SS1 -> X20TB1F13.SS; SL -> X20BM11k.SL1]
  Supervision = off
X20DOF322_108 : X20DOF322 v1.5.0.0  [SS1 -> X20TB1F10.SS; SL -> X20BM11i.SL1]
  Supervision = off
X20DOF322_206 : X20DOF322 v1.5.0.0  [SS1 -> X20TB1F18.SS; SL -> X20BM11ab.SL1]
  Supervision = off
X20DOF322_207 : X20DOF322 v1.5.0.0  [SS1 -> X20TB1F19.SS; SL -> X20BM11ac.SL1]
  Supervision = off
X20DOF322_208 : X20DOF322 v1.5.0.0  [SS1 -> X20TB1F20.SS; SL -> X20BM11ad.SL1]
  Supervision = off
X20MK0211 : X20MK0211 v1.0.0.3  [SL -> X20SL8100.SL1]
X20SC0402 : X20SC0402 v1.10.9.0  [SS1 -> X20TB52a.SS; SS2 -> X20TB52b.SS; SL -> X20BM33a.SL1]
  Supervision = off
  DigitalOutput01 =   // via SafeLogic works without PLC main and Direct works with it. Enable Transport signal is controlled via Safe Logic
  DigitalOutput02 = viaSafeLOGIC  // via SafeLogic works without PLC main and Direct works with it
X20SI8110_117 : X20SI8110 v1.10.9.0  [SS1 -> X20TB52c.SS; SL -> X20BM13.SL1]
  Supervision = off
  SafeModuleID = 3
X20SI8110_217 : X20SI8110 v1.10.9.0  [SS1 -> X20TB52e.SS; SL -> X20BM13a.SL1]
  Supervision = off
  SafeModuleID = 5
X20SL8100 : X20SL8100 v1.10.7.0  [PLK1 -> X20CP1382.IF3 (NodeNumber=10) [Cable Type=PowerlinkCable, Length=10, Version=1.0.0.3]; PLK2 -> 8AC114.60-2a.PLK1 (NodeNumber=10) [Cable Type=PowerlinkCable, Length=10, Version=1.0.0.3]; SS1 -> X20TB52.SS]
  Supervision = off
  SafeProject = EFI
  SafeDesigner = 4.3.4.4
  UnsafeInputINTs = 2
X20SM1436_007 : X20SM1436 v2.3.0.0  [SS1 -> X20TB12u.SS; SL -> X20BM31.SL1]
  Supervision = off
  DelayedCurrentSwitchOff01 = 5
  HoldingCurrent = 30
  RatedCurrent = 100
  MaximumCurrent = 110
  SM_SCALE_LOAD_UNITS_r1 = 2500
X20SM1436_008 : X20SM1436 v2.3.0.0  [SS1 -> X20TB12v.SS; SL -> X20BM31a.SL1]
  Supervision = off
  HoldingCurrent = 30
  RatedCurrent = 100
  MaximumCurrent = 110
  SM_SCALE_LOAD_UNITS_r1 = 2500
X20SO2110_118 : X20SO2110 v1.10.9.0  [SS1 -> X20TB52d.SS; SL -> X20BM33b.SL1]
  Supervision = off
  SafeModuleID = 4
X20SO2110_218 : X20SO2110 v1.10.9.0  [SS1 -> X20TB52f.SS; SL -> X20BM33c.SL1]
  Supervision = off
  SafeModuleID = 6
X20TB12 : X20TB12 v1.0.0.0
X20TB12a : X20TB12 v1.0.0.0
X20TB12b : X20TB12 v1.0.0.0
X20TB12c : X20TB12 v1.0.0.0
X20TB12d : X20TB12 v1.0.0.0
X20TB12e : X20TB12 v1.0.0.0
X20TB12f : X20TB12 v1.0.0.0
X20TB12g : X20TB12 v1.0.0.0
X20TB12h : X20TB12 v1.0.0.0
X20TB12i : X20TB12 v1.0.0.0
X20TB12j : X20TB12 v1.0.0.0
X20TB12k : X20TB12 v1.0.0.0 (Disabled=true)
X20TB12l : X20TB12 v1.0.0.0 (Disabled=true)
X20TB12m : X20TB12 v1.0.0.0 (Disabled=true)
X20TB12n : X20TB12 v1.0.0.0 (Disabled=true)
X20TB12o : X20TB12 v1.0.0.0
X20TB12p : X20TB12 v1.0.0.0
X20TB12q : X20TB12 v1.0.0.0
X20TB12r : X20TB12 v1.0.0.0
X20TB12s : X20TB12 v1.0.0.0
X20TB12t : X20TB12 v1.0.0.0
X20TB12u : X20TB12 v1.0.0.0
X20TB12v : X20TB12 v1.0.0.0
X20TB1F : X20TB1F v1.0.0.0
X20TB1F1 : X20TB1F v1.0.0.0
X20TB1F10 : X20TB1F v1.0.0.0
X20TB1F11 : X20TB1F v1.0.0.0
X20TB1F12 : X20TB1F v1.0.0.0
X20TB1F13 : X20TB1F v1.0.0.0
X20TB1F14 : X20TB1F v1.0.0.0
X20TB1F15 : X20TB1F v1.0.0.0
X20TB1F16 : X20TB1F v1.0.0.0
X20TB1F17 : X20TB1F v1.0.0.0
X20TB1F18 : X20TB1F v1.0.0.0
X20TB1F19 : X20TB1F v1.0.0.0
X20TB1F2 : X20TB1F v1.0.0.0
X20TB1F20 : X20TB1F v1.0.0.0
X20TB1F21 : X20TB1F v1.0.0.0
X20TB1F22 : X20TB1F v1.0.0.0
X20TB1F23 : X20TB1F v1.0.0.0
X20TB1F3 : X20TB1F v1.0.0.0
X20TB1F4 : X20TB1F v1.0.0.0
X20TB1F5 : X20TB1F v1.0.0.0
X20TB1F6 : X20TB1F v1.0.0.0
X20TB1F7 : X20TB1F v1.0.0.0
X20TB1F8 : X20TB1F v1.0.0.0
X20TB1F9 : X20TB1F v1.0.0.0
X20TB52 : X20TB52 v1.0.0.2
X20TB52a : X20TB52 v1.0.0.2
X20TB52b : X20TB52 v1.0.0.2
X20TB52c : X20TB52 v1.0.0.2
X20TB52d : X20TB52 v1.0.0.2
X20TB52e : X20TB52 v1.0.0.2
X20TB52f : X20TB52 v1.0.0.2
```
